// TwinCAT 3 PLC project plc_polycap_01
// ProgramVersion: 3.1.4023.0
// libraries:
//   LCLS General, * (SLAC)
//   lcls-twincat-motion, * (SLAC)
//   Tc2_Standard, * (Beckhoff Automation GmbH)
//   Tc2_System, * (Beckhoff Automation GmbH)
//   Tc3_Module, * (Beckhoff Automation GmbH)
// project tree:
//   GVLs/ Main.TcGVL
//   / PlcTask.TcTTO (not stored)
//   POUs/ PRG_SPEC.TcPOU
// real-time tasks:
//   TASK PlcTask: cycle T#10ms, priority 20, ADS port 350
// motion (NC):
//   TASK NC-Task 1 SAF: cycle T#2ms, priority 4, ADS port 501
//   TASK NC-Task 1 SVB: cycle T#10ms, priority 8, ADS port 511
//   AXIS Axis 1 POLYCAP-DET-Z (id 1)
//     Velo: Maximum=5
//     OtherSettings: AllowMotionCmdToSlave=true
//     encoder EncType=4
//       EncPara: ScaleFactorNumerator=7.8125e-05, MaxCount=#x0000ffff
//         Inc: RefSoftSyncMask=#x0000ffff
//     drive DrvType=24
//       Analog: VeloReferenz=10, TorqueSetpointScale=10, ScaleFactorActTorque=0.1
//       TimeComp: TaskDelayCycles=1
//     controller CtrType=1
//       CtrPara: PriorControlFactor=1
//         Observer: BandWidth=20
//   AXIS Axis 2 POLYCAP-CRY-N-SWI (id 2)
//     Velo: Maximum=5
//     OtherSettings: AllowMotionCmdToSlave=true
//     encoder EncType=4
//       EncPara: ScaleFactorNumerator=5.234375e-05, MaxCount=#x0000ffff
//         Inc: RefSoftSyncMask=#x0000ffff
//     drive DrvType=24
//       Analog: VeloReferenz=6.7, TorqueSetpointScale=10, ScaleFactorActTorque=0.1
//       TimeComp: TaskDelayCycles=1
//     controller CtrType=1
//       CtrPara: PriorControlFactor=1
//         Observer: BandWidth=20
//   AXIS Axis 3 POLYCAP-CRY-N-X (id 3)
//     Velo: Maximum=5
//     OtherSettings: AllowMotionCmdToSlave=true
//     encoder EncType=4
//       EncPara: ScaleFactorNumerator=7.8125e-05, MaxCount=#x0000ffff
//         Inc: RefSoftSyncMask=#x0000ffff
//     drive DrvType=24
//       Analog: VeloReferenz=10, TorqueSetpointScale=10, ScaleFactorActTorque=0.1
//       TimeComp: TaskDelayCycles=1
//     controller CtrType=1
//       CtrPara: PriorControlFactor=1
//         Observer: BandWidth=20
//   AXIS Axis 4 POLYCAP-CRY-N-ROT (id 4)
//     Velo: Maximum=5
//     OtherSettings: AllowMotionCmdToSlave=true
//     encoder EncType=4
//       EncPara: ScaleFactorNumerator=0.00015625, MaxCount=#x0000ffff
//         Inc: RefSoftSyncMask=#x0000ffff
//     drive DrvType=24
//       Analog: VeloReferenz=20, TorqueSetpointScale=10, ScaleFactorActTorque=0.1
//       TimeComp: TaskDelayCycles=1
//     controller CtrType=1
//       CtrPara: PriorControlFactor=1
//         Observer: BandWidth=20
//   AXIS Axis 5 POLYCAP-CRY-N-Y (id 5)
//     Velo: Maximum=5
//     OtherSettings: AllowMotionCmdToSlave=true
//     encoder EncType=4
//       EncPara: ScaleFactorNumerator=7.8125e-05, MaxCount=#x0000ffff
//         Inc: RefSoftSyncMask=#x0000ffff
//     drive DrvType=24
//       Analog: VeloReferenz=10, TorqueSetpointScale=10, ScaleFactorActTorque=0.1
//       TimeComp: TaskDelayCycles=1
//     controller CtrType=1
//       CtrPara: PriorControlFactor=1
//         Observer: BandWidth=20
//   AXIS Axis 6 POLYCAP-PC-N-X (id 6)
//     Velo: Maximum=5
//     OtherSettings: AllowMotionCmdToSlave=true
//     encoder EncType=4
//       EncPara: ScaleFactorNumerator=3.90625e-05, MaxCount=#x0000ffff
//         Inc: RefSoftSyncMask=#x0000ffff
//     drive DrvType=24
//       Analog: VeloReferenz=5, TorqueSetpointScale=10, ScaleFactorActTorque=0.1
//       TimeComp: TaskDelayCycles=1
//     controller CtrType=1
//       CtrPara: PriorControlFactor=1
//         Observer: BandWidth=20
//   AXIS Axis 7 POLYCAP-PC-N-Z (id 7)
//     Velo: Maximum=5
//     OtherSettings: AllowMotionCmdToSlave=true
//     encoder EncType=4
//       EncPara: ScaleFactorNumerator=1.953125e-05, MaxCount=#x0000ffff
//         Inc: RefSoftSyncMask=#x0000ffff
//     drive DrvType=24
//       Analog: VeloReferenz=2.5, TorqueSetpointScale=10, ScaleFactorActTorque=0.1
//       TimeComp: TaskDelayCycles=1
//     controller CtrType=1
//       CtrPara: PriorControlFactor=1
//         Observer: BandWidth=20
//   AXIS Axis 8 POLYCAP-PC-N-Y (id 8)
//     Velo: Maximum=5
//     OtherSettings: AllowMotionCmdToSlave=true
//     encoder EncType=4
//       EncPara: ScaleFactorNumerator=3.90625e-05, MaxCount=#x0000ffff
//         Inc: RefSoftSyncMask=#x0000ffff
//     drive DrvType=24
//       Analog: VeloReferenz=5, TorqueSetpointScale=10, ScaleFactorActTorque=0.1
//       TimeComp: TaskDelayCycles=1
//     controller CtrType=1
//       CtrPara: PriorControlFactor=1
//         Observer: BandWidth=20
//   AXIS Axis 9 POLYCAP-CRY-S-SWI (id 9)
//     Velo: Maximum=5
//     OtherSettings: AllowMotionCmdToSlave=true
//     encoder EncType=4
//       EncPara: ScaleFactorNumerator=5.234375e-05, MaxCount=#x0000ffff
//         Inc: RefSoftSyncMask=#x0000ffff
//     drive DrvType=24
//       Analog: VeloReferenz=6.7, TorqueSetpointScale=10, ScaleFactorActTorque=0.1
//       TimeComp: TaskDelayCycles=1
//     controller CtrType=1
//       CtrPara: PriorControlFactor=1
//         Observer: BandWidth=20
//   AXIS Axis 10 POLYCAP-CRY-S-X (id 10)
//     Velo: Maximum=5
//     OtherSettings: AllowMotionCmdToSlave=true
//     encoder EncType=4
//       EncPara: ScaleFactorNumerator=7.8125e-05, MaxCount=#x0000ffff
//         Inc: RefSoftSyncMask=#x0000ffff
//     drive DrvType=24
//       Analog: VeloReferenz=10, TorqueSetpointScale=10, ScaleFactorActTorque=0.1
//       TimeComp: TaskDelayCycles=1
//     controller CtrType=1
//       CtrPara: PriorControlFactor=1
//         Observer: BandWidth=20
//   AXIS Axis 11 POLYCAP-CRY-M-SWI (id 11)
//     Velo: Maximum=5
//     OtherSettings: AllowMotionCmdToSlave=true
//     encoder EncType=4
//       EncPara: ScaleFactorNumerator=5.234375e-05, MaxCount=#x0000ffff
//         Inc: RefSoftSyncMask=#x0000ffff
//     drive DrvType=24
//       Analog: VeloReferenz=6.7, TorqueSetpointScale=10, ScaleFactorActTorque=0.1
//       TimeComp: TaskDelayCycles=1
//     controller CtrType=1
//       CtrPara: PriorControlFactor=1
//         Observer: BandWidth=20
//   AXIS Axis 12 POLYCAP-CRY-M-X (id 12)
//     Velo: Maximum=5
//     OtherSettings: AllowMotionCmdToSlave=true
//     encoder EncType=4
//       EncPara: ScaleFactorNumerator=7.8125e-05, MaxCount=#x0000ffff
//         Inc: RefSoftSyncMask=#x0000ffff
//     drive DrvType=24
//       Analog: VeloReferenz=10, TorqueSetpointScale=10, ScaleFactorActTorque=0.1
//       TimeComp: TaskDelayCycles=1
//     controller CtrType=1
//       CtrPara: PriorControlFactor=1
//         Observer: BandWidth=20
//   AXIS Axis 13 POLYCAP-CRY-S-ROT (id 13)
//     Velo: Maximum=5
//     OtherSettings: AllowMotionCmdToSlave=true
//     encoder EncType=4
//       EncPara: ScaleFactorNumerator=0.00015625, MaxCount=#x0000ffff
//         Inc: RefSoftSyncMask=#x0000ffff
//     drive DrvType=24
//       Analog: VeloReferenz=20, TorqueSetpointScale=10, ScaleFactorActTorque=0.1
//       TimeComp: TaskDelayCycles=1
//     controller CtrType=1
//       CtrPara: PriorControlFactor=1
//         Observer: BandWidth=20
//   AXIS Axis 14 POLYCAP-CRY-S-Y (id 14)
//     Velo: Maximum=5
//     OtherSettings: AllowMotionCmdToSlave=true
//     encoder EncType=4
//       EncPara: ScaleFactorNumerator=7.8125e-05, MaxCount=#x0000ffff
//         Inc: RefSoftSyncMask=#x0000ffff
//     drive DrvType=24
//       Analog: VeloReferenz=10, TorqueSetpointScale=10, ScaleFactorActTorque=0.1
//       TimeComp: TaskDelayCycles=1
//     controller CtrType=1
//       CtrPara: PriorControlFactor=1
//         Observer: BandWidth=20
//   AXIS Axis 15 POLYCAP-CRY-M-ROT (id 15)
//     Velo: Maximum=5
//     OtherSettings: AllowMotionCmdToSlave=true
//     encoder EncType=4
//       EncPara: ScaleFactorNumerator=0.00015625, MaxCount=#x0000ffff
//         Inc: RefSoftSyncMask=#x0000ffff
//     drive DrvType=24
//       Analog: VeloReferenz=20, TorqueSetpointScale=10, ScaleFactorActTorque=0.1
//       TimeComp: TaskDelayCycles=1
//     controller CtrType=1
//       CtrPara: PriorControlFactor=1
//         Observer: BandWidth=20
//   AXIS Axis 16 POLYCAP-CRY-M-Y (id 16)
//     Velo: Maximum=5
//     OtherSettings: AllowMotionCmdToSlave=true
//     encoder EncType=4
//       EncPara: ScaleFactorNumerator=7.8125e-05, MaxCount=#x0000ffff
//         Inc: RefSoftSyncMask=#x0000ffff
//     drive DrvType=24
//       Analog: VeloReferenz=10, TorqueSetpointScale=10, ScaleFactorActTorque=0.1
//       TimeComp: TaskDelayCycles=1
//     controller CtrType=1
//       CtrPara: PriorControlFactor=1
//         Observer: BandWidth=20
//   AXIS Axis 17 POLYCAP-PC-S-X (id 17)
//     Velo: Maximum=5
//     OtherSettings: AllowMotionCmdToSlave=true
//     encoder EncType=4
//       EncPara: ScaleFactorNumerator=3.90625e-05, MaxCount=#x0000ffff
//         Inc: RefSoftSyncMask=#x0000ffff
//     drive DrvType=24
//       Analog: VeloReferenz=5, TorqueSetpointScale=10, ScaleFactorActTorque=0.1
//       TimeComp: TaskDelayCycles=1
//     controller CtrType=1
//       CtrPara: PriorControlFactor=1
//         Observer: BandWidth=20
//   AXIS Axis 18 POLYCAP-PC-S-Z (id 18)
//     Velo: Maximum=5
//     OtherSettings: AllowMotionCmdToSlave=true
//     encoder EncType=4
//       EncPara: ScaleFactorNumerator=1.953125e-05, MaxCount=#x0000ffff
//         Inc: RefSoftSyncMask=#x0000ffff
//     drive DrvType=24
//       Analog: VeloReferenz=2.5, TorqueSetpointScale=10, ScaleFactorActTorque=0.1
//       TimeComp: TaskDelayCycles=1
//     controller CtrType=1
//       CtrPara: PriorControlFactor=1
//         Observer: BandWidth=20
//   AXIS Axis 19 POLYCAP-PC-M-X (id 19)
//     Velo: Maximum=5
//     OtherSettings: AllowMotionCmdToSlave=true
//     encoder EncType=4
//       EncPara: ScaleFactorNumerator=3.90625e-05, MaxCount=#x0000ffff
//         Inc: RefSoftSyncMask=#x0000ffff
//     drive DrvType=24
//       Analog: VeloReferenz=5, TorqueSetpointScale=10, ScaleFactorActTorque=0.1
//       TimeComp: TaskDelayCycles=1
//     controller CtrType=1
//       CtrPara: PriorControlFactor=1
//         Observer: BandWidth=20
//   AXIS Axis 20 POLYCAP-PC-M-Z (id 20)
//     Velo: Maximum=5
//     OtherSettings: AllowMotionCmdToSlave=true
//     encoder EncType=4
//       EncPara: ScaleFactorNumerator=1.953125e-05, MaxCount=#x0000ffff
//         Inc: RefSoftSyncMask=#x0000ffff
//     drive DrvType=24
//       Analog: VeloReferenz=2.5, TorqueSetpointScale=10, ScaleFactorActTorque=0.1
//       TimeComp: TaskDelayCycles=1
//     controller CtrType=1
//       CtrPara: PriorControlFactor=1
//         Observer: BandWidth=20
//   AXIS Axis 21 POLYCAP-PC-S-Y (id 21)
//     Velo: Maximum=5
//     OtherSettings: AllowMotionCmdToSlave=true
//     encoder EncType=4
//       EncPara: ScaleFactorNumerator=3.90625e-05, MaxCount=#x0000ffff
//         Inc: RefSoftSyncMask=#x0000ffff
//     drive DrvType=24
//       Analog: VeloReferenz=5, TorqueSetpointScale=10, ScaleFactorActTorque=0.1
//       TimeComp: TaskDelayCycles=1
//     controller CtrType=1
//       CtrPara: PriorControlFactor=1
//         Observer: BandWidth=20
//   AXIS Axis 22 POLYCAP-PC-M-Y (id 22)
//     Velo: Maximum=5
//     OtherSettings: AllowMotionCmdToSlave=true
//     encoder EncType=4
//       EncPara: ScaleFactorNumerator=3.90625e-05, MaxCount=#x0000ffff
//         Inc: RefSoftSyncMask=#x0000ffff
//     drive DrvType=24
//       Analog: VeloReferenz=5, TorqueSetpointScale=10, ScaleFactorActTorque=0.1
//       TimeComp: TaskDelayCycles=1
//     controller CtrType=1
//       CtrPara: PriorControlFactor=1
//         Observer: BandWidth=20
// I/O:
//   DEVICE Device 1 (EtherCAT), AmsNetId 172.21.148.88.2.1
//     Term 1 (EK1200) [EK1200-5000 EtherCAT Power supply (2A E-Bus)]
//       POLYCAP1-EL7031-E1 [EL7031 1Ch. Stepper motor output stage (24V, 1.5A)]
//       Term 3 (EL6070) [EL6070 1Ch. Licensing-Terminal]
//       Term 4 (EL7031) [EL7031 1Ch. Stepper motor output stage (24V, 1.5A)]
//       POLYCAP1-EL1088-E4 [EL1088 8Ch. Dig. Input 24V, 3ms, negative]
//       Term 6 (EL7031) [EL7031 1Ch. Stepper motor output stage (24V, 1.5A)]
//       Term 7 (EL7031) [EL7031 1Ch. Stepper motor output stage (24V, 1.5A)]
//       Term 8 (EL7031) [EL7031 1Ch. Stepper motor output stage (24V, 1.5A)]
//       Term 9 (EL7031) [EL7031 1Ch. Stepper motor output stage (24V, 1.5A)]
//       POLYCAP1-EL1088-E9 [EL1088 8Ch. Dig. Input 24V, 3ms, negative]
//       Term 11 (EK1122) [EK1122 2 port EtherCAT junction]
//         Term 12 (EK1100) [EK1100 EtherCAT Coupler (2A E-Bus)]
//           Term 13 (EL7031) [EL7031 1Ch. Stepper motor output stage (24V, 1.5A)]
//           Term 14 (EL7031) [EL7031 1Ch. Stepper motor output stage (24V, 1.5A)]
//           POLYCAP2-EL1088-E3 [EL1088 8Ch. Dig. Input 24V, 3ms, negative]
//           Term 16 (EL7031) [EL7031 1Ch. Stepper motor output stage (24V, 1.5A)]
//           Term 17 (EL7031) [EL7031 1Ch. Stepper motor output stage (24V, 1.5A)]
//           Term 18 (EL7031) [EL7031 1Ch. Stepper motor output stage (24V, 1.5A)]
//           Term 19 (EL7031) [EL7031 1Ch. Stepper motor output stage (24V, 1.5A)]
//           POLYCAP2-EL1088-E8 [EL1088 8Ch. Dig. Input 24V, 3ms, negative]
//           Term 21 (EL7031) [EL7031 1Ch. Stepper motor output stage (24V, 1.5A)]
//           Term 22 (EL7031) [EL7031 1Ch. Stepper motor output stage (24V, 1.5A)]
//           Term 23 (EL9410) [EL9410 E-Bus Power Supplier  (Diagnostics)]
//           Term 24 (EL7031) [EL7031 1Ch. Stepper motor output stage (24V, 1.5A)]
//           Term 25 (EL7031) [EL7031 1Ch. Stepper motor output stage (24V, 1.5A)]
//           POLYCAP2-EL1088-E14 [EL1088 8Ch. Dig. Input 24V, 3ms, negative]
//           Term 27 (EL7031) [EL7031 1Ch. Stepper motor output stage (24V, 1.5A)]
//           Term 28 (EL7031) [EL7031 1Ch. Stepper motor output stage (24V, 1.5A)]
//           Term 29 (EL7031) [EL7031 1Ch. Stepper motor output stage (24V, 1.5A)]
//           Term 30 (EL7031) [EL7031 1Ch. Stepper motor output stage (24V, 1.5A)]
//           POLYCAP2-EL1088-E19 [EL1088 8Ch. Dig. Input 24V, 3ms, negative]
//           Term 32 (EL7031) [EL7031 1Ch. Stepper motor output stage (24V, 1.5A)]
//           Term 33 (EL7031) [EL7031 1Ch. Stepper motor output stage (24V, 1.5A)]
//           Term 34 (EL9011)
// variable links:
//   (this object) <-> Device 1 (EtherCAT)/Term 1 (EK1200)/POLYCAP1-EL7031-E1
//     Drive/Inputs/In/nState1 @bit 3 <-> STM Status/Status/Error
//     Drive/Inputs/In/nState1 @bit 5 <-> STM Status/Status/Moving negative
//     Drive/Inputs/In/nState1 @bit 4 <-> STM Status/Status/Moving positive
//     Drive/Inputs/In/nState1 @bit 1 <-> STM Status/Status/Ready
//     Drive/Inputs/In/nState1 <-> STM Status/Status/Ready to enable
//     Drive/Inputs/In/nState1 @bit 6 <-> STM Status/Status/Torque reduced
//     Drive/Inputs/In/nState1 @bit 2 <-> STM Status/Status/Warning
//     Drive/Inputs/In/nState2 @bit 3 <-> STM Status/Status/Digital input 1
//     Drive/Inputs/In/nState2 @bit 4 <-> STM Status/Status/Digital input 2
//     Drive/Inputs/In/nState2 @bit 5 <-> STM Status/Status/Sync error
//     Drive/Inputs/In/nState2 @bit 7 <-> STM Status/Status/TxPDO Toggle
//     Drive/Inputs/In/nState4 @bit 1 <-> WcState/InputToggle
//     Drive/Inputs/In/nState4 <-> WcState/WcState
//     Drive/Outputs/Out/nCtrl1 <-> STM Control/Control/Enable
//     Drive/Outputs/Out/nCtrl1 @bit 2 <-> STM Control/Control/Reduce torque
//     Drive/Outputs/Out/nCtrl1 @bit 1 <-> STM Control/Control/Reset
//     Drive/Outputs/Out/nDataOut2[0] <-> STM Velocity/Velocity
//     Enc/Inputs/In/nDataIn1[0] <-> ENC Status compact/Counter value
//     Enc/Inputs/In/nDataIn2[0] <-> ENC Status compact/Latch value
//     Enc/Inputs/In/nState1 @bit 4 <-> ENC Status compact/Status/Counter overflow
//     Enc/Inputs/In/nState1 @bit 3 <-> ENC Status compact/Status/Counter underflow
//     Enc/Inputs/In/nState1 @bit 1 <-> ENC Status compact/Status/Latch extern valid
//     Enc/Inputs/In/nState1 @bit 2 <-> ENC Status compact/Status/Set counter done
//     Enc/Inputs/In/nState2 @bit 4 <-> ENC Status compact/Status/Status of extern latch
//     Enc/Inputs/In/nState2 @bit 5 <-> ENC Status compact/Status/Sync error
//     Enc/Inputs/In/nState2 @bit 7 <-> ENC Status compact/Status/TxPDO Toggle
//     Enc/Inputs/In/nState4 @bit 1 <-> WcState/InputToggle
//     Enc/Inputs/In/nState4 <-> WcState/WcState
//     Enc/Outputs/Out/nCtrl1 @bit 3 <-> ENC Control compact/Control/Enable latch extern on negative edge
//     Enc/Outputs/Out/nCtrl1 @bit 1 <-> ENC Control compact/Control/Enable latch extern on positive edge
//     Enc/Outputs/Out/nCtrl1 @bit 2 <-> ENC Control compact/Control/Set counter
//     Enc/Outputs/Out/nDataOut1[0] <-> ENC Control compact/Set counter value
//   (this object) <-> Device 1 (EtherCAT)/Term 1 (EK1200)/Term 4 (EL7031)
//     Drive/Inputs/In/nState1 @bit 3 <-> STM Status/Status/Error
//     Drive/Inputs/In/nState1 @bit 5 <-> STM Status/Status/Moving negative
//     Drive/Inputs/In/nState1 @bit 4 <-> STM Status/Status/Moving positive
//     Drive/Inputs/In/nState1 @bit 1 <-> STM Status/Status/Ready
//     Drive/Inputs/In/nState1 <-> STM Status/Status/Ready to enable
//     Drive/Inputs/In/nState1 @bit 6 <-> STM Status/Status/Torque reduced
//     Drive/Inputs/In/nState1 @bit 2 <-> STM Status/Status/Warning
//     Drive/Inputs/In/nState2 @bit 3 <-> STM Status/Status/Digital input 1
//     Drive/Inputs/In/nState2 @bit 4 <-> STM Status/Status/Digital input 2
//     Drive/Inputs/In/nState2 @bit 5 <-> STM Status/Status/Sync error
//     Drive/Inputs/In/nState2 @bit 7 <-> STM Status/Status/TxPDO Toggle
//     Drive/Inputs/In/nState4 @bit 1 <-> WcState/InputToggle
//     Drive/Inputs/In/nState4 <-> WcState/WcState
//     Drive/Outputs/Out/nCtrl1 <-> STM Control/Control/Enable
//     Drive/Outputs/Out/nCtrl1 @bit 2 <-> STM Control/Control/Reduce torque
//     Drive/Outputs/Out/nCtrl1 @bit 1 <-> STM Control/Control/Reset
//     Drive/Outputs/Out/nDataOut2[0] <-> STM Velocity/Velocity
//     Enc/Inputs/In/nDataIn1[0] <-> ENC Status compact/Counter value
//     Enc/Inputs/In/nDataIn2[0] <-> ENC Status compact/Latch value
//     Enc/Inputs/In/nState1 @bit 4 <-> ENC Status compact/Status/Counter overflow
//     Enc/Inputs/In/nState1 @bit 3 <-> ENC Status compact/Status/Counter underflow
//     Enc/Inputs/In/nState1 @bit 1 <-> ENC Status compact/Status/Latch extern valid
//     Enc/Inputs/In/nState1 @bit 2 <-> ENC Status compact/Status/Set counter done
//     Enc/Inputs/In/nState2 @bit 4 <-> ENC Status compact/Status/Status of extern latch
//     Enc/Inputs/In/nState2 @bit 5 <-> ENC Status compact/Status/Sync error
//     Enc/Inputs/In/nState2 @bit 7 <-> ENC Status compact/Status/TxPDO Toggle
//     Enc/Inputs/In/nState4 @bit 1 <-> WcState/InputToggle
//     Enc/Inputs/In/nState4 <-> WcState/WcState
//     Enc/Outputs/Out/nCtrl1 @bit 3 <-> ENC Control compact/Control/Enable latch extern on negative edge
//     Enc/Outputs/Out/nCtrl1 @bit 1 <-> ENC Control compact/Control/Enable latch extern on positive edge
//     Enc/Outputs/Out/nCtrl1 @bit 2 <-> ENC Control compact/Control/Set counter
//     Enc/Outputs/Out/nDataOut1[0] <-> ENC Control compact/Set counter value
//   (this object) <-> Device 1 (EtherCAT)/Term 1 (EK1200)/Term 6 (EL7031)
//     Drive/Inputs/In/nState1 @bit 3 <-> STM Status/Status/Error
//     Drive/Inputs/In/nState1 @bit 5 <-> STM Status/Status/Moving negative
//     Drive/Inputs/In/nState1 @bit 4 <-> STM Status/Status/Moving positive
//     Drive/Inputs/In/nState1 @bit 1 <-> STM Status/Status/Ready
//     Drive/Inputs/In/nState1 <-> STM Status/Status/Ready to enable
//     Drive/Inputs/In/nState1 @bit 6 <-> STM Status/Status/Torque reduced
//     Drive/Inputs/In/nState1 @bit 2 <-> STM Status/Status/Warning
//     Drive/Inputs/In/nState2 @bit 3 <-> STM Status/Status/Digital input 1
//     Drive/Inputs/In/nState2 @bit 4 <-> STM Status/Status/Digital input 2
//     Drive/Inputs/In/nState2 @bit 5 <-> STM Status/Status/Sync error
//     Drive/Inputs/In/nState2 @bit 7 <-> STM Status/Status/TxPDO Toggle
//     Drive/Inputs/In/nState4 @bit 1 <-> WcState/InputToggle
//     Drive/Inputs/In/nState4 <-> WcState/WcState
//     Drive/Outputs/Out/nCtrl1 <-> STM Control/Control/Enable
//     Drive/Outputs/Out/nCtrl1 @bit 2 <-> STM Control/Control/Reduce torque
//     Drive/Outputs/Out/nCtrl1 @bit 1 <-> STM Control/Control/Reset
//     Drive/Outputs/Out/nDataOut2[0] <-> STM Velocity/Velocity
//     Enc/Inputs/In/nDataIn1[0] <-> ENC Status compact/Counter value
//     Enc/Inputs/In/nDataIn2[0] <-> ENC Status compact/Latch value
//     Enc/Inputs/In/nState1 @bit 4 <-> ENC Status compact/Status/Counter overflow
//     Enc/Inputs/In/nState1 @bit 3 <-> ENC Status compact/Status/Counter underflow
//     Enc/Inputs/In/nState1 @bit 1 <-> ENC Status compact/Status/Latch extern valid
//     Enc/Inputs/In/nState1 @bit 2 <-> ENC Status compact/Status/Set counter done
//     Enc/Inputs/In/nState2 @bit 4 <-> ENC Status compact/Status/Status of extern latch
//     Enc/Inputs/In/nState2 @bit 5 <-> ENC Status compact/Status/Sync error
//     Enc/Inputs/In/nState2 @bit 7 <-> ENC Status compact/Status/TxPDO Toggle
//     Enc/Inputs/In/nState4 @bit 1 <-> WcState/InputToggle
//     Enc/Inputs/In/nState4 <-> WcState/WcState
//     Enc/Outputs/Out/nCtrl1 @bit 3 <-> ENC Control compact/Control/Enable latch extern on negative edge
//     Enc/Outputs/Out/nCtrl1 @bit 1 <-> ENC Control compact/Control/Enable latch extern on positive edge
//     Enc/Outputs/Out/nCtrl1 @bit 2 <-> ENC Control compact/Control/Set counter
//     Enc/Outputs/Out/nDataOut1[0] <-> ENC Control compact/Set counter value
//   (this object) <-> Device 1 (EtherCAT)/Term 1 (EK1200)/Term 7 (EL7031)
//     Drive/Inputs/In/nState1 @bit 3 <-> STM Status/Status/Error
//     Drive/Inputs/In/nState1 @bit 5 <-> STM Status/Status/Moving negative
//     Drive/Inputs/In/nState1 @bit 4 <-> STM Status/Status/Moving positive
//     Drive/Inputs/In/nState1 @bit 1 <-> STM Status/Status/Ready
//     Drive/Inputs/In/nState1 <-> STM Status/Status/Ready to enable
//     Drive/Inputs/In/nState1 @bit 6 <-> STM Status/Status/Torque reduced
//     Drive/Inputs/In/nState1 @bit 2 <-> STM Status/Status/Warning
//     Drive/Inputs/In/nState2 @bit 3 <-> STM Status/Status/Digital input 1
//     Drive/Inputs/In/nState2 @bit 4 <-> STM Status/Status/Digital input 2
//     Drive/Inputs/In/nState2 @bit 5 <-> STM Status/Status/Sync error
//     Drive/Inputs/In/nState2 @bit 7 <-> STM Status/Status/TxPDO Toggle
//     Drive/Inputs/In/nState4 @bit 1 <-> WcState/InputToggle
//     Drive/Inputs/In/nState4 <-> WcState/WcState
//     Drive/Outputs/Out/nCtrl1 <-> STM Control/Control/Enable
//     Drive/Outputs/Out/nCtrl1 @bit 2 <-> STM Control/Control/Reduce torque
//     Drive/Outputs/Out/nCtrl1 @bit 1 <-> STM Control/Control/Reset
//     Drive/Outputs/Out/nDataOut2[0] <-> STM Velocity/Velocity
//     Enc/Inputs/In/nDataIn1[0] <-> ENC Status compact/Counter value
//     Enc/Inputs/In/nDataIn2[0] <-> ENC Status compact/Latch value
//     Enc/Inputs/In/nState1 @bit 4 <-> ENC Status compact/Status/Counter overflow
//     Enc/Inputs/In/nState1 @bit 3 <-> ENC Status compact/Status/Counter underflow
//     Enc/Inputs/In/nState1 @bit 1 <-> ENC Status compact/Status/Latch extern valid
//     Enc/Inputs/In/nState1 @bit 2 <-> ENC Status compact/Status/Set counter done
//     Enc/Inputs/In/nState2 @bit 4 <-> ENC Status compact/Status/Status of extern latch
//     Enc/Inputs/In/nState2 @bit 5 <-> ENC Status compact/Status/Sync error
//     Enc/Inputs/In/nState2 @bit 7 <-> ENC Status compact/Status/TxPDO Toggle
//     Enc/Inputs/In/nState4 @bit 1 <-> WcState/InputToggle
//     Enc/Inputs/In/nState4 <-> WcState/WcState
//     Enc/Outputs/Out/nCtrl1 @bit 3 <-> ENC Control compact/Control/Enable latch extern on negative edge
//     Enc/Outputs/Out/nCtrl1 @bit 1 <-> ENC Control compact/Control/Enable latch extern on positive edge
//     Enc/Outputs/Out/nCtrl1 @bit 2 <-> ENC Control compact/Control/Set counter
//     Enc/Outputs/Out/nDataOut1[0] <-> ENC Control compact/Set counter value
//   (this object) <-> Device 1 (EtherCAT)/Term 1 (EK1200)/Term 8 (EL7031)
//     Drive/Inputs/In/nState1 @bit 3 <-> STM Status/Status/Error
//     Drive/Inputs/In/nState1 @bit 5 <-> STM Status/Status/Moving negative
//     Drive/Inputs/In/nState1 @bit 4 <-> STM Status/Status/Moving positive
//     Drive/Inputs/In/nState1 @bit 1 <-> STM Status/Status/Ready
//     Drive/Inputs/In/nState1 <-> STM Status/Status/Ready to enable
//     Drive/Inputs/In/nState1 @bit 6 <-> STM Status/Status/Torque reduced
//     Drive/Inputs/In/nState1 @bit 2 <-> STM Status/Status/Warning
//     Drive/Inputs/In/nState2 @bit 3 <-> STM Status/Status/Digital input 1
//     Drive/Inputs/In/nState2 @bit 4 <-> STM Status/Status/Digital input 2
//     Drive/Inputs/In/nState2 @bit 5 <-> STM Status/Status/Sync error
//     Drive/Inputs/In/nState2 @bit 7 <-> STM Status/Status/TxPDO Toggle
//     Drive/Inputs/In/nState4 @bit 1 <-> WcState/InputToggle
//     Drive/Inputs/In/nState4 <-> WcState/WcState
//     Drive/Outputs/Out/nCtrl1 <-> STM Control/Control/Enable
//     Drive/Outputs/Out/nCtrl1 @bit 2 <-> STM Control/Control/Reduce torque
//     Drive/Outputs/Out/nCtrl1 @bit 1 <-> STM Control/Control/Reset
//     Drive/Outputs/Out/nDataOut2[0] <-> STM Velocity/Velocity
//     Enc/Inputs/In/nDataIn1[0] <-> ENC Status compact/Counter value
//     Enc/Inputs/In/nDataIn2[0] <-> ENC Status compact/Latch value
//     Enc/Inputs/In/nState1 @bit 4 <-> ENC Status compact/Status/Counter overflow
//     Enc/Inputs/In/nState1 @bit 3 <-> ENC Status compact/Status/Counter underflow
//     Enc/Inputs/In/nState1 @bit 1 <-> ENC Status compact/Status/Latch extern valid
//     Enc/Inputs/In/nState1 @bit 2 <-> ENC Status compact/Status/Set counter done
//     Enc/Inputs/In/nState2 @bit 4 <-> ENC Status compact/Status/Status of extern latch
//     Enc/Inputs/In/nState2 @bit 5 <-> ENC Status compact/Status/Sync error
//     Enc/Inputs/In/nState2 @bit 7 <-> ENC Status compact/Status/TxPDO Toggle
//     Enc/Inputs/In/nState4 @bit 1 <-> WcState/InputToggle
//     Enc/Inputs/In/nState4 <-> WcState/WcState
//     Enc/Outputs/Out/nCtrl1 @bit 3 <-> ENC Control compact/Control/Enable latch extern on negative edge
//     Enc/Outputs/Out/nCtrl1 @bit 1 <-> ENC Control compact/Control/Enable latch extern on positive edge
//     Enc/Outputs/Out/nCtrl1 @bit 2 <-> ENC Control compact/Control/Set counter
//     Enc/Outputs/Out/nDataOut1[0] <-> ENC Control compact/Set counter value
//   (this object) <-> Device 1 (EtherCAT)/Term 1 (EK1200)/Term 9 (EL7031)
//     Drive/Inputs/In/nState1 @bit 3 <-> STM Status/Status/Error
//     Drive/Inputs/In/nState1 @bit 5 <-> STM Status/Status/Moving negative
//     Drive/Inputs/In/nState1 @bit 4 <-> STM Status/Status/Moving positive
//     Drive/Inputs/In/nState1 @bit 1 <-> STM Status/Status/Ready
//     Drive/Inputs/In/nState1 <-> STM Status/Status/Ready to enable
//     Drive/Inputs/In/nState1 @bit 6 <-> STM Status/Status/Torque reduced
//     Drive/Inputs/In/nState1 @bit 2 <-> STM Status/Status/Warning
//     Drive/Inputs/In/nState2 @bit 3 <-> STM Status/Status/Digital input 1
//     Drive/Inputs/In/nState2 @bit 4 <-> STM Status/Status/Digital input 2
//     Drive/Inputs/In/nState2 @bit 5 <-> STM Status/Status/Sync error
//     Drive/Inputs/In/nState2 @bit 7 <-> STM Status/Status/TxPDO Toggle
//     Drive/Inputs/In/nState4 @bit 1 <-> WcState/InputToggle
//     Drive/Inputs/In/nState4 <-> WcState/WcState
//     Drive/Outputs/Out/nCtrl1 <-> STM Control/Control/Enable
//     Drive/Outputs/Out/nCtrl1 @bit 2 <-> STM Control/Control/Reduce torque
//     Drive/Outputs/Out/nCtrl1 @bit 1 <-> STM Control/Control/Reset
//     Drive/Outputs/Out/nDataOut2[0] <-> STM Velocity/Velocity
//     Enc/Inputs/In/nDataIn1[0] <-> ENC Status compact/Counter value
//     Enc/Inputs/In/nDataIn2[0] <-> ENC Status compact/Latch value
//     Enc/Inputs/In/nState1 @bit 4 <-> ENC Status compact/Status/Counter overflow
//     Enc/Inputs/In/nState1 @bit 3 <-> ENC Status compact/Status/Counter underflow
//     Enc/Inputs/In/nState1 @bit 1 <-> ENC Status compact/Status/Latch extern valid
//     Enc/Inputs/In/nState1 @bit 2 <-> ENC Status compact/Status/Set counter done
//     Enc/Inputs/In/nState2 @bit 4 <-> ENC Status compact/Status/Status of extern latch
//     Enc/Inputs/In/nState2 @bit 5 <-> ENC Status compact/Status/Sync error
//     Enc/Inputs/In/nState2 @bit 7 <-> ENC Status compact/Status/TxPDO Toggle
//     Enc/Inputs/In/nState4 @bit 1 <-> WcState/InputToggle
//     Enc/Inputs/In/nState4 <-> WcState/WcState
//     Enc/Outputs/Out/nCtrl1 @bit 3 <-> ENC Control compact/Control/Enable latch extern on negative edge
//     Enc/Outputs/Out/nCtrl1 @bit 1 <-> ENC Control compact/Control/Enable latch extern on positive edge
//     Enc/Outputs/Out/nCtrl1 @bit 2 <-> ENC Control compact/Control/Set counter
//     Enc/Outputs/Out/nDataOut1[0] <-> ENC Control compact/Set counter value
//   (this object) <-> Device 1 (EtherCAT)/Term 1 (EK1200)/Term 11 (EK1122)/Term 12 (EK1100)/Term 13 (EL7031)
//     Drive/Inputs/In/nState1 @bit 3 <-> STM Status/Status/Error
//     Drive/Inputs/In/nState1 @bit 5 <-> STM Status/Status/Moving negative
//     Drive/Inputs/In/nState1 @bit 4 <-> STM Status/Status/Moving positive
//     Drive/Inputs/In/nState1 @bit 1 <-> STM Status/Status/Ready
//     Drive/Inputs/In/nState1 <-> STM Status/Status/Ready to enable
//     Drive/Inputs/In/nState1 @bit 6 <-> STM Status/Status/Torque reduced
//     Drive/Inputs/In/nState1 @bit 2 <-> STM Status/Status/Warning
//     Drive/Inputs/In/nState2 @bit 3 <-> STM Status/Status/Digital input 1
//     Drive/Inputs/In/nState2 @bit 4 <-> STM Status/Status/Digital input 2
//     Drive/Inputs/In/nState2 @bit 5 <-> STM Status/Status/Sync error
//     Drive/Inputs/In/nState2 @bit 7 <-> STM Status/Status/TxPDO Toggle
//     Drive/Inputs/In/nState4 @bit 1 <-> WcState/InputToggle
//     Drive/Inputs/In/nState4 <-> WcState/WcState
//     Drive/Outputs/Out/nCtrl1 <-> STM Control/Control/Enable
//     Drive/Outputs/Out/nCtrl1 @bit 2 <-> STM Control/Control/Reduce torque
//     Drive/Outputs/Out/nCtrl1 @bit 1 <-> STM Control/Control/Reset
//     Drive/Outputs/Out/nDataOut2[0] <-> STM Velocity/Velocity
//     Enc/Inputs/In/nDataIn1[0] <-> ENC Status compact/Counter value
//     Enc/Inputs/In/nDataIn2[0] <-> ENC Status compact/Latch value
//     Enc/Inputs/In/nState1 @bit 4 <-> ENC Status compact/Status/Counter overflow
//     Enc/Inputs/In/nState1 @bit 3 <-> ENC Status compact/Status/Counter underflow
//     Enc/Inputs/In/nState1 @bit 1 <-> ENC Status compact/Status/Latch extern valid
//     Enc/Inputs/In/nState1 @bit 2 <-> ENC Status compact/Status/Set counter done
//     Enc/Inputs/In/nState2 @bit 4 <-> ENC Status compact/Status/Status of extern latch
//     Enc/Inputs/In/nState2 @bit 5 <-> ENC Status compact/Status/Sync error
//     Enc/Inputs/In/nState2 @bit 7 <-> ENC Status compact/Status/TxPDO Toggle
//     Enc/Inputs/In/nState4 @bit 1 <-> WcState/InputToggle
//     Enc/Inputs/In/nState4 <-> WcState/WcState
//     Enc/Outputs/Out/nCtrl1 @bit 3 <-> ENC Control compact/Control/Enable latch extern on negative edge
//     Enc/Outputs/Out/nCtrl1 @bit 1 <-> ENC Control compact/Control/Enable latch extern on positive edge
//     Enc/Outputs/Out/nCtrl1 @bit 2 <-> ENC Control compact/Control/Set counter
//     Enc/Outputs/Out/nDataOut1[0] <-> ENC Control compact/Set counter value
//   (this object) <-> Device 1 (EtherCAT)/Term 1 (EK1200)/Term 11 (EK1122)/Term 12 (EK1100)/Term 14 (EL7031)
//     Drive/Inputs/In/nState1 @bit 3 <-> STM Status/Status/Error
//     Drive/Inputs/In/nState1 @bit 5 <-> STM Status/Status/Moving negative
//     Drive/Inputs/In/nState1 @bit 4 <-> STM Status/Status/Moving positive
//     Drive/Inputs/In/nState1 @bit 1 <-> STM Status/Status/Ready
//     Drive/Inputs/In/nState1 <-> STM Status/Status/Ready to enable
//     Drive/Inputs/In/nState1 @bit 6 <-> STM Status/Status/Torque reduced
//     Drive/Inputs/In/nState1 @bit 2 <-> STM Status/Status/Warning
//     Drive/Inputs/In/nState2 @bit 3 <-> STM Status/Status/Digital input 1
//     Drive/Inputs/In/nState2 @bit 4 <-> STM Status/Status/Digital input 2
//     Drive/Inputs/In/nState2 @bit 5 <-> STM Status/Status/Sync error
//     Drive/Inputs/In/nState2 @bit 7 <-> STM Status/Status/TxPDO Toggle
//     Drive/Inputs/In/nState4 @bit 1 <-> WcState/InputToggle
//     Drive/Inputs/In/nState4 <-> WcState/WcState
//     Drive/Outputs/Out/nCtrl1 <-> STM Control/Control/Enable
//     Drive/Outputs/Out/nCtrl1 @bit 2 <-> STM Control/Control/Reduce torque
//     Drive/Outputs/Out/nCtrl1 @bit 1 <-> STM Control/Control/Reset
//     Drive/Outputs/Out/nDataOut2[0] <-> STM Velocity/Velocity
//     Enc/Inputs/In/nDataIn1[0] <-> ENC Status compact/Counter value
//     Enc/Inputs/In/nDataIn2[0] <-> ENC Status compact/Latch value
//     Enc/Inputs/In/nState1 @bit 4 <-> ENC Status compact/Status/Counter overflow
//     Enc/Inputs/In/nState1 @bit 3 <-> ENC Status compact/Status/Counter underflow
//     Enc/Inputs/In/nState1 @bit 1 <-> ENC Status compact/Status/Latch extern valid
//     Enc/Inputs/In/nState1 @bit 2 <-> ENC Status compact/Status/Set counter done
//     Enc/Inputs/In/nState2 @bit 4 <-> ENC Status compact/Status/Status of extern latch
//     Enc/Inputs/In/nState2 @bit 5 <-> ENC Status compact/Status/Sync error
//     Enc/Inputs/In/nState2 @bit 7 <-> ENC Status compact/Status/TxPDO Toggle
//     Enc/Inputs/In/nState4 @bit 1 <-> WcState/InputToggle
//     Enc/Inputs/In/nState4 <-> WcState/WcState
//     Enc/Outputs/Out/nCtrl1 @bit 3 <-> ENC Control compact/Control/Enable latch extern on negative edge
//     Enc/Outputs/Out/nCtrl1 @bit 1 <-> ENC Control compact/Control/Enable latch extern on positive edge
//     Enc/Outputs/Out/nCtrl1 @bit 2 <-> ENC Control compact/Control/Set counter
//     Enc/Outputs/Out/nDataOut1[0] <-> ENC Control compact/Set counter value
//   (this object) <-> Device 1 (EtherCAT)/Term 1 (EK1200)/Term 11 (EK1122)/Term 12 (EK1100)/Term 16 (EL7031)
//     Drive/Inputs/In/nState1 @bit 3 <-> STM Status/Status/Error
//     Drive/Inputs/In/nState1 @bit 5 <-> STM Status/Status/Moving negative
//     Drive/Inputs/In/nState1 @bit 4 <-> STM Status/Status/Moving positive
//     Drive/Inputs/In/nState1 @bit 1 <-> STM Status/Status/Ready
//     Drive/Inputs/In/nState1 <-> STM Status/Status/Ready to enable
//     Drive/Inputs/In/nState1 @bit 6 <-> STM Status/Status/Torque reduced
//     Drive/Inputs/In/nState1 @bit 2 <-> STM Status/Status/Warning
//     Drive/Inputs/In/nState2 @bit 3 <-> STM Status/Status/Digital input 1
//     Drive/Inputs/In/nState2 @bit 4 <-> STM Status/Status/Digital input 2
//     Drive/Inputs/In/nState2 @bit 5 <-> STM Status/Status/Sync error
//     Drive/Inputs/In/nState2 @bit 7 <-> STM Status/Status/TxPDO Toggle
//     Drive/Inputs/In/nState4 @bit 1 <-> WcState/InputToggle
//     Drive/Inputs/In/nState4 <-> WcState/WcState
//     Drive/Outputs/Out/nCtrl1 <-> STM Control/Control/Enable
//     Drive/Outputs/Out/nCtrl1 @bit 2 <-> STM Control/Control/Reduce torque
//     Drive/Outputs/Out/nCtrl1 @bit 1 <-> STM Control/Control/Reset
//     Drive/Outputs/Out/nDataOut2[0] <-> STM Velocity/Velocity
//     Enc/Inputs/In/nDataIn1[0] <-> ENC Status compact/Counter value
//     Enc/Inputs/In/nDataIn2[0] <-> ENC Status compact/Latch value
//     Enc/Inputs/In/nState1 @bit 4 <-> ENC Status compact/Status/Counter overflow
//     Enc/Inputs/In/nState1 @bit 3 <-> ENC Status compact/Status/Counter underflow
//     Enc/Inputs/In/nState1 @bit 1 <-> ENC Status compact/Status/Latch extern valid
//     Enc/Inputs/In/nState1 @bit 2 <-> ENC Status compact/Status/Set counter done
//     Enc/Inputs/In/nState2 @bit 4 <-> ENC Status compact/Status/Status of extern latch
//     Enc/Inputs/In/nState2 @bit 5 <-> ENC Status compact/Status/Sync error
//     Enc/Inputs/In/nState2 @bit 7 <-> ENC Status compact/Status/TxPDO Toggle
//     Enc/Inputs/In/nState4 @bit 1 <-> WcState/InputToggle
//     Enc/Inputs/In/nState4 <-> WcState/WcState
//     Enc/Outputs/Out/nCtrl1 @bit 3 <-> ENC Control compact/Control/Enable latch extern on negative edge
//     Enc/Outputs/Out/nCtrl1 @bit 1 <-> ENC Control compact/Control/Enable latch extern on positive edge
//     Enc/Outputs/Out/nCtrl1 @bit 2 <-> ENC Control compact/Control/Set counter
//     Enc/Outputs/Out/nDataOut1[0] <-> ENC Control compact/Set counter value
//   (this object) <-> Device 1 (EtherCAT)/Term 1 (EK1200)/Term 11 (EK1122)/Term 12 (EK1100)/Term 17 (EL7031)
//     Drive/Inputs/In/nState1 @bit 3 <-> STM Status/Status/Error
//     Drive/Inputs/In/nState1 @bit 5 <-> STM Status/Status/Moving negative
//     Drive/Inputs/In/nState1 @bit 4 <-> STM Status/Status/Moving positive
//     Drive/Inputs/In/nState1 @bit 1 <-> STM Status/Status/Ready
//     Drive/Inputs/In/nState1 <-> STM Status/Status/Ready to enable
//     Drive/Inputs/In/nState1 @bit 6 <-> STM Status/Status/Torque reduced
//     Drive/Inputs/In/nState1 @bit 2 <-> STM Status/Status/Warning
//     Drive/Inputs/In/nState2 @bit 3 <-> STM Status/Status/Digital input 1
//     Drive/Inputs/In/nState2 @bit 4 <-> STM Status/Status/Digital input 2
//     Drive/Inputs/In/nState2 @bit 5 <-> STM Status/Status/Sync error
//     Drive/Inputs/In/nState2 @bit 7 <-> STM Status/Status/TxPDO Toggle
//     Drive/Inputs/In/nState4 @bit 1 <-> WcState/InputToggle
//     Drive/Inputs/In/nState4 <-> WcState/WcState
//     Drive/Outputs/Out/nCtrl1 <-> STM Control/Control/Enable
//     Drive/Outputs/Out/nCtrl1 @bit 2 <-> STM Control/Control/Reduce torque
//     Drive/Outputs/Out/nCtrl1 @bit 1 <-> STM Control/Control/Reset
//     Drive/Outputs/Out/nDataOut2[0] <-> STM Velocity/Velocity
//     Enc/Inputs/In/nDataIn1[0] <-> ENC Status compact/Counter value
//     Enc/Inputs/In/nDataIn2[0] <-> ENC Status compact/Latch value
//     Enc/Inputs/In/nState1 @bit 4 <-> ENC Status compact/Status/Counter overflow
//     Enc/Inputs/In/nState1 @bit 3 <-> ENC Status compact/Status/Counter underflow
//     Enc/Inputs/In/nState1 @bit 1 <-> ENC Status compact/Status/Latch extern valid
//     Enc/Inputs/In/nState1 @bit 2 <-> ENC Status compact/Status/Set counter done
//     Enc/Inputs/In/nState2 @bit 4 <-> ENC Status compact/Status/Status of extern latch
//     Enc/Inputs/In/nState2 @bit 5 <-> ENC Status compact/Status/Sync error
//     Enc/Inputs/In/nState2 @bit 7 <-> ENC Status compact/Status/TxPDO Toggle
//     Enc/Inputs/In/nState4 @bit 1 <-> WcState/InputToggle
//     Enc/Inputs/In/nState4 <-> WcState/WcState
//     Enc/Outputs/Out/nCtrl1 @bit 3 <-> ENC Control compact/Control/Enable latch extern on negative edge
//     Enc/Outputs/Out/nCtrl1 @bit 1 <-> ENC Control compact/Control/Enable latch extern on positive edge
//     Enc/Outputs/Out/nCtrl1 @bit 2 <-> ENC Control compact/Control/Set counter
//     Enc/Outputs/Out/nDataOut1[0] <-> ENC Control compact/Set counter value
//   (this object) <-> Device 1 (EtherCAT)/Term 1 (EK1200)/Term 11 (EK1122)/Term 12 (EK1100)/Term 18 (EL7031)
//     Drive/Inputs/In/nState1 @bit 3 <-> STM Status/Status/Error
//     Drive/Inputs/In/nState1 @bit 5 <-> STM Status/Status/Moving negative
//     Drive/Inputs/In/nState1 @bit 4 <-> STM Status/Status/Moving positive
//     Drive/Inputs/In/nState1 @bit 1 <-> STM Status/Status/Ready
//     Drive/Inputs/In/nState1 <-> STM Status/Status/Ready to enable
//     Drive/Inputs/In/nState1 @bit 6 <-> STM Status/Status/Torque reduced
//     Drive/Inputs/In/nState1 @bit 2 <-> STM Status/Status/Warning
//     Drive/Inputs/In/nState2 @bit 3 <-> STM Status/Status/Digital input 1
//     Drive/Inputs/In/nState2 @bit 4 <-> STM Status/Status/Digital input 2
//     Drive/Inputs/In/nState2 @bit 5 <-> STM Status/Status/Sync error
//     Drive/Inputs/In/nState2 @bit 7 <-> STM Status/Status/TxPDO Toggle
//     Drive/Inputs/In/nState4 @bit 1 <-> WcState/InputToggle
//     Drive/Inputs/In/nState4 <-> WcState/WcState
//     Drive/Outputs/Out/nCtrl1 <-> STM Control/Control/Enable
//     Drive/Outputs/Out/nCtrl1 @bit 2 <-> STM Control/Control/Reduce torque
//     Drive/Outputs/Out/nCtrl1 @bit 1 <-> STM Control/Control/Reset
//     Drive/Outputs/Out/nDataOut2[0] <-> STM Velocity/Velocity
//     Enc/Inputs/In/nDataIn1[0] <-> ENC Status compact/Counter value
//     Enc/Inputs/In/nDataIn2[0] <-> ENC Status compact/Latch value
//     Enc/Inputs/In/nState1 @bit 4 <-> ENC Status compact/Status/Counter overflow
//     Enc/Inputs/In/nState1 @bit 3 <-> ENC Status compact/Status/Counter underflow
//     Enc/Inputs/In/nState1 @bit 1 <-> ENC Status compact/Status/Latch extern valid
//     Enc/Inputs/In/nState1 @bit 2 <-> ENC Status compact/Status/Set counter done
//     Enc/Inputs/In/nState2 @bit 4 <-> ENC Status compact/Status/Status of extern latch
//     Enc/Inputs/In/nState2 @bit 5 <-> ENC Status compact/Status/Sync error
//     Enc/Inputs/In/nState2 @bit 7 <-> ENC Status compact/Status/TxPDO Toggle
//     Enc/Inputs/In/nState4 @bit 1 <-> WcState/InputToggle
//     Enc/Inputs/In/nState4 <-> WcState/WcState
//     Enc/Outputs/Out/nCtrl1 @bit 3 <-> ENC Control compact/Control/Enable latch extern on negative edge
//     Enc/Outputs/Out/nCtrl1 @bit 1 <-> ENC Control compact/Control/Enable latch extern on positive edge
//     Enc/Outputs/Out/nCtrl1 @bit 2 <-> ENC Control compact/Control/Set counter
//     Enc/Outputs/Out/nDataOut1[0] <-> ENC Control compact/Set counter value
//   (this object) <-> Device 1 (EtherCAT)/Term 1 (EK1200)/Term 11 (EK1122)/Term 12 (EK1100)/Term 19 (EL7031)
//     Drive/Inputs/In/nState1 @bit 3 <-> STM Status/Status/Error
//     Drive/Inputs/In/nState1 @bit 5 <-> STM Status/Status/Moving negative
//     Drive/Inputs/In/nState1 @bit 4 <-> STM Status/Status/Moving positive
//     Drive/Inputs/In/nState1 @bit 1 <-> STM Status/Status/Ready
//     Drive/Inputs/In/nState1 <-> STM Status/Status/Ready to enable
//     Drive/Inputs/In/nState1 @bit 6 <-> STM Status/Status/Torque reduced
//     Drive/Inputs/In/nState1 @bit 2 <-> STM Status/Status/Warning
//     Drive/Inputs/In/nState2 @bit 3 <-> STM Status/Status/Digital input 1
//     Drive/Inputs/In/nState2 @bit 4 <-> STM Status/Status/Digital input 2
//     Drive/Inputs/In/nState2 @bit 5 <-> STM Status/Status/Sync error
//     Drive/Inputs/In/nState2 @bit 7 <-> STM Status/Status/TxPDO Toggle
//     Drive/Inputs/In/nState4 @bit 1 <-> WcState/InputToggle
//     Drive/Inputs/In/nState4 <-> WcState/WcState
//     Drive/Outputs/Out/nCtrl1 <-> STM Control/Control/Enable
//     Drive/Outputs/Out/nCtrl1 @bit 2 <-> STM Control/Control/Reduce torque
//     Drive/Outputs/Out/nCtrl1 @bit 1 <-> STM Control/Control/Reset
//     Drive/Outputs/Out/nDataOut2[0] <-> STM Velocity/Velocity
//     Enc/Inputs/In/nDataIn1[0] <-> ENC Status compact/Counter value
//     Enc/Inputs/In/nDataIn2[0] <-> ENC Status compact/Latch value
//     Enc/Inputs/In/nState1 @bit 4 <-> ENC Status compact/Status/Counter overflow
//     Enc/Inputs/In/nState1 @bit 3 <-> ENC Status compact/Status/Counter underflow
//     Enc/Inputs/In/nState1 @bit 1 <-> ENC Status compact/Status/Latch extern valid
//     Enc/Inputs/In/nState1 @bit 2 <-> ENC Status compact/Status/Set counter done
//     Enc/Inputs/In/nState2 @bit 4 <-> ENC Status compact/Status/Status of extern latch
//     Enc/Inputs/In/nState2 @bit 5 <-> ENC Status compact/Status/Sync error
//     Enc/Inputs/In/nState2 @bit 7 <-> ENC Status compact/Status/TxPDO Toggle
//     Enc/Inputs/In/nState4 @bit 1 <-> WcState/InputToggle
//     Enc/Inputs/In/nState4 <-> WcState/WcState
//     Enc/Outputs/Out/nCtrl1 @bit 3 <-> ENC Control compact/Control/Enable latch extern on negative edge
//     Enc/Outputs/Out/nCtrl1 @bit 1 <-> ENC Control compact/Control/Enable latch extern on positive edge
//     Enc/Outputs/Out/nCtrl1 @bit 2 <-> ENC Control compact/Control/Set counter
//     Enc/Outputs/Out/nDataOut1[0] <-> ENC Control compact/Set counter value
//   (this object) <-> Device 1 (EtherCAT)/Term 1 (EK1200)/Term 11 (EK1122)/Term 12 (EK1100)/Term 21 (EL7031)
//     Drive/Inputs/In/nState1 @bit 3 <-> STM Status/Status/Error
//     Drive/Inputs/In/nState1 @bit 5 <-> STM Status/Status/Moving negative
//     Drive/Inputs/In/nState1 @bit 4 <-> STM Status/Status/Moving positive
//     Drive/Inputs/In/nState1 @bit 1 <-> STM Status/Status/Ready
//     Drive/Inputs/In/nState1 <-> STM Status/Status/Ready to enable
//     Drive/Inputs/In/nState1 @bit 6 <-> STM Status/Status/Torque reduced
//     Drive/Inputs/In/nState1 @bit 2 <-> STM Status/Status/Warning
//     Drive/Inputs/In/nState2 @bit 3 <-> STM Status/Status/Digital input 1
//     Drive/Inputs/In/nState2 @bit 4 <-> STM Status/Status/Digital input 2
//     Drive/Inputs/In/nState2 @bit 5 <-> STM Status/Status/Sync error
//     Drive/Inputs/In/nState2 @bit 7 <-> STM Status/Status/TxPDO Toggle
//     Drive/Inputs/In/nState4 @bit 1 <-> WcState/InputToggle
//     Drive/Inputs/In/nState4 <-> WcState/WcState
//     Drive/Outputs/Out/nCtrl1 <-> STM Control/Control/Enable
//     Drive/Outputs/Out/nCtrl1 @bit 2 <-> STM Control/Control/Reduce torque
//     Drive/Outputs/Out/nCtrl1 @bit 1 <-> STM Control/Control/Reset
//     Drive/Outputs/Out/nDataOut2[0] <-> STM Velocity/Velocity
//     Enc/Inputs/In/nDataIn1[0] <-> ENC Status compact/Counter value
//     Enc/Inputs/In/nDataIn2[0] <-> ENC Status compact/Latch value
//     Enc/Inputs/In/nState1 @bit 4 <-> ENC Status compact/Status/Counter overflow
//     Enc/Inputs/In/nState1 @bit 3 <-> ENC Status compact/Status/Counter underflow
//     Enc/Inputs/In/nState1 @bit 1 <-> ENC Status compact/Status/Latch extern valid
//     Enc/Inputs/In/nState1 @bit 2 <-> ENC Status compact/Status/Set counter done
//     Enc/Inputs/In/nState2 @bit 4 <-> ENC Status compact/Status/Status of extern latch
//     Enc/Inputs/In/nState2 @bit 5 <-> ENC Status compact/Status/Sync error
//     Enc/Inputs/In/nState2 @bit 7 <-> ENC Status compact/Status/TxPDO Toggle
//     Enc/Inputs/In/nState4 @bit 1 <-> WcState/InputToggle
//     Enc/Inputs/In/nState4 <-> WcState/WcState
//     Enc/Outputs/Out/nCtrl1 @bit 3 <-> ENC Control compact/Control/Enable latch extern on negative edge
//     Enc/Outputs/Out/nCtrl1 @bit 1 <-> ENC Control compact/Control/Enable latch extern on positive edge
//     Enc/Outputs/Out/nCtrl1 @bit 2 <-> ENC Control compact/Control/Set counter
//     Enc/Outputs/Out/nDataOut1[0] <-> ENC Control compact/Set counter value
//   (this object) <-> Device 1 (EtherCAT)/Term 1 (EK1200)/Term 11 (EK1122)/Term 12 (EK1100)/Term 22 (EL7031)
//     Drive/Inputs/In/nState1 @bit 3 <-> STM Status/Status/Error
//     Drive/Inputs/In/nState1 @bit 5 <-> STM Status/Status/Moving negative
//     Drive/Inputs/In/nState1 @bit 4 <-> STM Status/Status/Moving positive
//     Drive/Inputs/In/nState1 @bit 1 <-> STM Status/Status/Ready
//     Drive/Inputs/In/nState1 <-> STM Status/Status/Ready to enable
//     Drive/Inputs/In/nState1 @bit 6 <-> STM Status/Status/Torque reduced
//     Drive/Inputs/In/nState1 @bit 2 <-> STM Status/Status/Warning
//     Drive/Inputs/In/nState2 @bit 3 <-> STM Status/Status/Digital input 1
//     Drive/Inputs/In/nState2 @bit 4 <-> STM Status/Status/Digital input 2
//     Drive/Inputs/In/nState2 @bit 5 <-> STM Status/Status/Sync error
//     Drive/Inputs/In/nState2 @bit 7 <-> STM Status/Status/TxPDO Toggle
//     Drive/Inputs/In/nState4 @bit 1 <-> WcState/InputToggle
//     Drive/Inputs/In/nState4 <-> WcState/WcState
//     Drive/Outputs/Out/nCtrl1 <-> STM Control/Control/Enable
//     Drive/Outputs/Out/nCtrl1 @bit 2 <-> STM Control/Control/Reduce torque
//     Drive/Outputs/Out/nCtrl1 @bit 1 <-> STM Control/Control/Reset
//     Drive/Outputs/Out/nDataOut2[0] <-> STM Velocity/Velocity
//     Enc/Inputs/In/nDataIn1[0] <-> ENC Status compact/Counter value
//     Enc/Inputs/In/nDataIn2[0] <-> ENC Status compact/Latch value
//     Enc/Inputs/In/nState1 @bit 4 <-> ENC Status compact/Status/Counter overflow
//     Enc/Inputs/In/nState1 @bit 3 <-> ENC Status compact/Status/Counter underflow
//     Enc/Inputs/In/nState1 @bit 1 <-> ENC Status compact/Status/Latch extern valid
//     Enc/Inputs/In/nState1 @bit 2 <-> ENC Status compact/Status/Set counter done
//     Enc/Inputs/In/nState2 @bit 4 <-> ENC Status compact/Status/Status of extern latch
//     Enc/Inputs/In/nState2 @bit 5 <-> ENC Status compact/Status/Sync error
//     Enc/Inputs/In/nState2 @bit 7 <-> ENC Status compact/Status/TxPDO Toggle
//     Enc/Inputs/In/nState4 @bit 1 <-> WcState/InputToggle
//     Enc/Inputs/In/nState4 <-> WcState/WcState
//     Enc/Outputs/Out/nCtrl1 @bit 3 <-> ENC Control compact/Control/Enable latch extern on negative edge
//     Enc/Outputs/Out/nCtrl1 @bit 1 <-> ENC Control compact/Control/Enable latch extern on positive edge
//     Enc/Outputs/Out/nCtrl1 @bit 2 <-> ENC Control compact/Control/Set counter
//     Enc/Outputs/Out/nDataOut1[0] <-> ENC Control compact/Set counter value
//   (this object) <-> Device 1 (EtherCAT)/Term 1 (EK1200)/Term 11 (EK1122)/Term 12 (EK1100)/Term 24 (EL7031)
//     Drive/Inputs/In/nState1 @bit 3 <-> STM Status/Status/Error
//     Drive/Inputs/In/nState1 @bit 5 <-> STM Status/Status/Moving negative
//     Drive/Inputs/In/nState1 @bit 4 <-> STM Status/Status/Moving positive
//     Drive/Inputs/In/nState1 @bit 1 <-> STM Status/Status/Ready
//     Drive/Inputs/In/nState1 <-> STM Status/Status/Ready to enable
//     Drive/Inputs/In/nState1 @bit 6 <-> STM Status/Status/Torque reduced
//     Drive/Inputs/In/nState1 @bit 2 <-> STM Status/Status/Warning
//     Drive/Inputs/In/nState2 @bit 3 <-> STM Status/Status/Digital input 1
//     Drive/Inputs/In/nState2 @bit 4 <-> STM Status/Status/Digital input 2
//     Drive/Inputs/In/nState2 @bit 5 <-> STM Status/Status/Sync error
//     Drive/Inputs/In/nState2 @bit 7 <-> STM Status/Status/TxPDO Toggle
//     Drive/Inputs/In/nState4 @bit 1 <-> WcState/InputToggle
//     Drive/Inputs/In/nState4 <-> WcState/WcState
//     Drive/Outputs/Out/nCtrl1 <-> STM Control/Control/Enable
//     Drive/Outputs/Out/nCtrl1 @bit 2 <-> STM Control/Control/Reduce torque
//     Drive/Outputs/Out/nCtrl1 @bit 1 <-> STM Control/Control/Reset
//     Drive/Outputs/Out/nDataOut2[0] <-> STM Velocity/Velocity
//     Enc/Inputs/In/nDataIn1[0] <-> ENC Status compact/Counter value
//     Enc/Inputs/In/nDataIn2[0] <-> ENC Status compact/Latch value
//     Enc/Inputs/In/nState1 @bit 4 <-> ENC Status compact/Status/Counter overflow
//     Enc/Inputs/In/nState1 @bit 3 <-> ENC Status compact/Status/Counter underflow
//     Enc/Inputs/In/nState1 @bit 1 <-> ENC Status compact/Status/Latch extern valid
//     Enc/Inputs/In/nState1 @bit 2 <-> ENC Status compact/Status/Set counter done
//     Enc/Inputs/In/nState2 @bit 4 <-> ENC Status compact/Status/Status of extern latch
//     Enc/Inputs/In/nState2 @bit 5 <-> ENC Status compact/Status/Sync error
//     Enc/Inputs/In/nState2 @bit 7 <-> ENC Status compact/Status/TxPDO Toggle
//     Enc/Inputs/In/nState4 @bit 1 <-> WcState/InputToggle
//     Enc/Inputs/In/nState4 <-> WcState/WcState
//     Enc/Outputs/Out/nCtrl1 @bit 3 <-> ENC Control compact/Control/Enable latch extern on negative edge
//     Enc/Outputs/Out/nCtrl1 @bit 1 <-> ENC Control compact/Control/Enable latch extern on positive edge
//     Enc/Outputs/Out/nCtrl1 @bit 2 <-> ENC Control compact/Control/Set counter
//     Enc/Outputs/Out/nDataOut1[0] <-> ENC Control compact/Set counter value
//   (this object) <-> Device 1 (EtherCAT)/Term 1 (EK1200)/Term 11 (EK1122)/Term 12 (EK1100)/Term 25 (EL7031)
//     Drive/Inputs/In/nState1 @bit 3 <-> STM Status/Status/Error
//     Drive/Inputs/In/nState1 @bit 5 <-> STM Status/Status/Moving negative
//     Drive/Inputs/In/nState1 @bit 4 <-> STM Status/Status/Moving positive
//     Drive/Inputs/In/nState1 @bit 1 <-> STM Status/Status/Ready
//     Drive/Inputs/In/nState1 <-> STM Status/Status/Ready to enable
//     Drive/Inputs/In/nState1 @bit 6 <-> STM Status/Status/Torque reduced
//     Drive/Inputs/In/nState1 @bit 2 <-> STM Status/Status/Warning
//     Drive/Inputs/In/nState2 @bit 3 <-> STM Status/Status/Digital input 1
//     Drive/Inputs/In/nState2 @bit 4 <-> STM Status/Status/Digital input 2
//     Drive/Inputs/In/nState2 @bit 5 <-> STM Status/Status/Sync error
//     Drive/Inputs/In/nState2 @bit 7 <-> STM Status/Status/TxPDO Toggle
//     Drive/Inputs/In/nState4 @bit 1 <-> WcState/InputToggle
//     Drive/Inputs/In/nState4 <-> WcState/WcState
//     Drive/Outputs/Out/nCtrl1 <-> STM Control/Control/Enable
//     Drive/Outputs/Out/nCtrl1 @bit 2 <-> STM Control/Control/Reduce torque
//     Drive/Outputs/Out/nCtrl1 @bit 1 <-> STM Control/Control/Reset
//     Drive/Outputs/Out/nDataOut2[0] <-> STM Velocity/Velocity
//     Enc/Inputs/In/nDataIn1[0] <-> ENC Status compact/Counter value
//     Enc/Inputs/In/nDataIn2[0] <-> ENC Status compact/Latch value
//     Enc/Inputs/In/nState1 @bit 4 <-> ENC Status compact/Status/Counter overflow
//     Enc/Inputs/In/nState1 @bit 3 <-> ENC Status compact/Status/Counter underflow
//     Enc/Inputs/In/nState1 @bit 1 <-> ENC Status compact/Status/Latch extern valid
//     Enc/Inputs/In/nState1 @bit 2 <-> ENC Status compact/Status/Set counter done
//     Enc/Inputs/In/nState2 @bit 4 <-> ENC Status compact/Status/Status of extern latch
//     Enc/Inputs/In/nState2 @bit 5 <-> ENC Status compact/Status/Sync error
//     Enc/Inputs/In/nState2 @bit 7 <-> ENC Status compact/Status/TxPDO Toggle
//     Enc/Inputs/In/nState4 @bit 1 <-> WcState/InputToggle
//     Enc/Inputs/In/nState4 <-> WcState/WcState
//     Enc/Outputs/Out/nCtrl1 @bit 3 <-> ENC Control compact/Control/Enable latch extern on negative edge
//     Enc/Outputs/Out/nCtrl1 @bit 1 <-> ENC Control compact/Control/Enable latch extern on positive edge
//     Enc/Outputs/Out/nCtrl1 @bit 2 <-> ENC Control compact/Control/Set counter
//     Enc/Outputs/Out/nDataOut1[0] <-> ENC Control compact/Set counter value
//   (this object) <-> Device 1 (EtherCAT)/Term 1 (EK1200)/Term 11 (EK1122)/Term 12 (EK1100)/Term 27 (EL7031)
//     Drive/Inputs/In/nState1 @bit 3 <-> STM Status/Status/Error
//     Drive/Inputs/In/nState1 @bit 5 <-> STM Status/Status/Moving negative
//     Drive/Inputs/In/nState1 @bit 4 <-> STM Status/Status/Moving positive
//     Drive/Inputs/In/nState1 @bit 1 <-> STM Status/Status/Ready
//     Drive/Inputs/In/nState1 <-> STM Status/Status/Ready to enable
//     Drive/Inputs/In/nState1 @bit 6 <-> STM Status/Status/Torque reduced
//     Drive/Inputs/In/nState1 @bit 2 <-> STM Status/Status/Warning
//     Drive/Inputs/In/nState2 @bit 3 <-> STM Status/Status/Digital input 1
//     Drive/Inputs/In/nState2 @bit 4 <-> STM Status/Status/Digital input 2
//     Drive/Inputs/In/nState2 @bit 5 <-> STM Status/Status/Sync error
//     Drive/Inputs/In/nState2 @bit 7 <-> STM Status/Status/TxPDO Toggle
//     Drive/Inputs/In/nState4 @bit 1 <-> WcState/InputToggle
//     Drive/Inputs/In/nState4 <-> WcState/WcState
//     Drive/Outputs/Out/nCtrl1 <-> STM Control/Control/Enable
//     Drive/Outputs/Out/nCtrl1 @bit 2 <-> STM Control/Control/Reduce torque
//     Drive/Outputs/Out/nCtrl1 @bit 1 <-> STM Control/Control/Reset
//     Drive/Outputs/Out/nDataOut2[0] <-> STM Velocity/Velocity
//     Enc/Inputs/In/nDataIn1[0] <-> ENC Status compact/Counter value
//     Enc/Inputs/In/nDataIn2[0] <-> ENC Status compact/Latch value
//     Enc/Inputs/In/nState1 @bit 4 <-> ENC Status compact/Status/Counter overflow
//     Enc/Inputs/In/nState1 @bit 3 <-> ENC Status compact/Status/Counter underflow
//     Enc/Inputs/In/nState1 @bit 1 <-> ENC Status compact/Status/Latch extern valid
//     Enc/Inputs/In/nState1 @bit 2 <-> ENC Status compact/Status/Set counter done
//     Enc/Inputs/In/nState2 @bit 4 <-> ENC Status compact/Status/Status of extern latch
//     Enc/Inputs/In/nState2 @bit 5 <-> ENC Status compact/Status/Sync error
//     Enc/Inputs/In/nState2 @bit 7 <-> ENC Status compact/Status/TxPDO Toggle
//     Enc/Inputs/In/nState4 @bit 1 <-> WcState/InputToggle
//     Enc/Inputs/In/nState4 <-> WcState/WcState
//     Enc/Outputs/Out/nCtrl1 @bit 3 <-> ENC Control compact/Control/Enable latch extern on negative edge
//     Enc/Outputs/Out/nCtrl1 @bit 1 <-> ENC Control compact/Control/Enable latch extern on positive edge
//     Enc/Outputs/Out/nCtrl1 @bit 2 <-> ENC Control compact/Control/Set counter
//     Enc/Outputs/Out/nDataOut1[0] <-> ENC Control compact/Set counter value
//   (this object) <-> Device 1 (EtherCAT)/Term 1 (EK1200)/Term 11 (EK1122)/Term 12 (EK1100)/Term 28 (EL7031)
//     Drive/Inputs/In/nState1 @bit 3 <-> STM Status/Status/Error
//     Drive/Inputs/In/nState1 @bit 5 <-> STM Status/Status/Moving negative
//     Drive/Inputs/In/nState1 @bit 4 <-> STM Status/Status/Moving positive
//     Drive/Inputs/In/nState1 @bit 1 <-> STM Status/Status/Ready
//     Drive/Inputs/In/nState1 <-> STM Status/Status/Ready to enable
//     Drive/Inputs/In/nState1 @bit 6 <-> STM Status/Status/Torque reduced
//     Drive/Inputs/In/nState1 @bit 2 <-> STM Status/Status/Warning
//     Drive/Inputs/In/nState2 @bit 3 <-> STM Status/Status/Digital input 1
//     Drive/Inputs/In/nState2 @bit 4 <-> STM Status/Status/Digital input 2
//     Drive/Inputs/In/nState2 @bit 5 <-> STM Status/Status/Sync error
//     Drive/Inputs/In/nState2 @bit 7 <-> STM Status/Status/TxPDO Toggle
//     Drive/Inputs/In/nState4 @bit 1 <-> WcState/InputToggle
//     Drive/Inputs/In/nState4 <-> WcState/WcState
//     Drive/Outputs/Out/nCtrl1 <-> STM Control/Control/Enable
//     Drive/Outputs/Out/nCtrl1 @bit 2 <-> STM Control/Control/Reduce torque
//     Drive/Outputs/Out/nCtrl1 @bit 1 <-> STM Control/Control/Reset
//     Drive/Outputs/Out/nDataOut2[0] <-> STM Velocity/Velocity
//     Enc/Inputs/In/nDataIn1[0] <-> ENC Status compact/Counter value
//     Enc/Inputs/In/nDataIn2[0] <-> ENC Status compact/Latch value
//     Enc/Inputs/In/nState1 @bit 4 <-> ENC Status compact/Status/Counter overflow
//     Enc/Inputs/In/nState1 @bit 3 <-> ENC Status compact/Status/Counter underflow
//     Enc/Inputs/In/nState1 @bit 1 <-> ENC Status compact/Status/Latch extern valid
//     Enc/Inputs/In/nState1 @bit 2 <-> ENC Status compact/Status/Set counter done
//     Enc/Inputs/In/nState2 @bit 4 <-> ENC Status compact/Status/Status of extern latch
//     Enc/Inputs/In/nState2 @bit 5 <-> ENC Status compact/Status/Sync error
//     Enc/Inputs/In/nState2 @bit 7 <-> ENC Status compact/Status/TxPDO Toggle
//     Enc/Inputs/In/nState4 @bit 1 <-> WcState/InputToggle
//     Enc/Inputs/In/nState4 <-> WcState/WcState
//     Enc/Outputs/Out/nCtrl1 @bit 3 <-> ENC Control compact/Control/Enable latch extern on negative edge
//     Enc/Outputs/Out/nCtrl1 @bit 1 <-> ENC Control compact/Control/Enable latch extern on positive edge
//     Enc/Outputs/Out/nCtrl1 @bit 2 <-> ENC Control compact/Control/Set counter
//     Enc/Outputs/Out/nDataOut1[0] <-> ENC Control compact/Set counter value
//   (this object) <-> Device 1 (EtherCAT)/Term 1 (EK1200)/Term 11 (EK1122)/Term 12 (EK1100)/Term 29 (EL7031)
//     Drive/Inputs/In/nState1 @bit 3 <-> STM Status/Status/Error
//     Drive/Inputs/In/nState1 @bit 5 <-> STM Status/Status/Moving negative
//     Drive/Inputs/In/nState1 @bit 4 <-> STM Status/Status/Moving positive
//     Drive/Inputs/In/nState1 @bit 1 <-> STM Status/Status/Ready
//     Drive/Inputs/In/nState1 <-> STM Status/Status/Ready to enable
//     Drive/Inputs/In/nState1 @bit 6 <-> STM Status/Status/Torque reduced
//     Drive/Inputs/In/nState1 @bit 2 <-> STM Status/Status/Warning
//     Drive/Inputs/In/nState2 @bit 3 <-> STM Status/Status/Digital input 1
//     Drive/Inputs/In/nState2 @bit 4 <-> STM Status/Status/Digital input 2
//     Drive/Inputs/In/nState2 @bit 5 <-> STM Status/Status/Sync error
//     Drive/Inputs/In/nState2 @bit 7 <-> STM Status/Status/TxPDO Toggle
//     Drive/Inputs/In/nState4 @bit 1 <-> WcState/InputToggle
//     Drive/Inputs/In/nState4 <-> WcState/WcState
//     Drive/Outputs/Out/nCtrl1 <-> STM Control/Control/Enable
//     Drive/Outputs/Out/nCtrl1 @bit 2 <-> STM Control/Control/Reduce torque
//     Drive/Outputs/Out/nCtrl1 @bit 1 <-> STM Control/Control/Reset
//     Drive/Outputs/Out/nDataOut2[0] <-> STM Velocity/Velocity
//     Enc/Inputs/In/nDataIn1[0] <-> ENC Status compact/Counter value
//     Enc/Inputs/In/nDataIn2[0] <-> ENC Status compact/Latch value
//     Enc/Inputs/In/nState1 @bit 4 <-> ENC Status compact/Status/Counter overflow
//     Enc/Inputs/In/nState1 @bit 3 <-> ENC Status compact/Status/Counter underflow
//     Enc/Inputs/In/nState1 @bit 1 <-> ENC Status compact/Status/Latch extern valid
//     Enc/Inputs/In/nState1 @bit 2 <-> ENC Status compact/Status/Set counter done
//     Enc/Inputs/In/nState2 @bit 4 <-> ENC Status compact/Status/Status of extern latch
//     Enc/Inputs/In/nState2 @bit 5 <-> ENC Status compact/Status/Sync error
//     Enc/Inputs/In/nState2 @bit 7 <-> ENC Status compact/Status/TxPDO Toggle
//     Enc/Inputs/In/nState4 @bit 1 <-> WcState/InputToggle
//     Enc/Inputs/In/nState4 <-> WcState/WcState
//     Enc/Outputs/Out/nCtrl1 @bit 3 <-> ENC Control compact/Control/Enable latch extern on negative edge
//     Enc/Outputs/Out/nCtrl1 @bit 1 <-> ENC Control compact/Control/Enable latch extern on positive edge
//     Enc/Outputs/Out/nCtrl1 @bit 2 <-> ENC Control compact/Control/Set counter
//     Enc/Outputs/Out/nDataOut1[0] <-> ENC Control compact/Set counter value
//   (this object) <-> Device 1 (EtherCAT)/Term 1 (EK1200)/Term 11 (EK1122)/Term 12 (EK1100)/Term 30 (EL7031)
//     Drive/Inputs/In/nState1 @bit 3 <-> STM Status/Status/Error
//     Drive/Inputs/In/nState1 @bit 5 <-> STM Status/Status/Moving negative
//     Drive/Inputs/In/nState1 @bit 4 <-> STM Status/Status/Moving positive
//     Drive/Inputs/In/nState1 @bit 1 <-> STM Status/Status/Ready
//     Drive/Inputs/In/nState1 <-> STM Status/Status/Ready to enable
//     Drive/Inputs/In/nState1 @bit 6 <-> STM Status/Status/Torque reduced
//     Drive/Inputs/In/nState1 @bit 2 <-> STM Status/Status/Warning
//     Drive/Inputs/In/nState2 @bit 3 <-> STM Status/Status/Digital input 1
//     Drive/Inputs/In/nState2 @bit 4 <-> STM Status/Status/Digital input 2
//     Drive/Inputs/In/nState2 @bit 5 <-> STM Status/Status/Sync error
//     Drive/Inputs/In/nState2 @bit 7 <-> STM Status/Status/TxPDO Toggle
//     Drive/Inputs/In/nState4 @bit 1 <-> WcState/InputToggle
//     Drive/Inputs/In/nState4 <-> WcState/WcState
//     Drive/Outputs/Out/nCtrl1 <-> STM Control/Control/Enable
//     Drive/Outputs/Out/nCtrl1 @bit 2 <-> STM Control/Control/Reduce torque
//     Drive/Outputs/Out/nCtrl1 @bit 1 <-> STM Control/Control/Reset
//     Drive/Outputs/Out/nDataOut2[0] <-> STM Velocity/Velocity
//     Enc/Inputs/In/nDataIn1[0] <-> ENC Status compact/Counter value
//     Enc/Inputs/In/nDataIn2[0] <-> ENC Status compact/Latch value
//     Enc/Inputs/In/nState1 @bit 4 <-> ENC Status compact/Status/Counter overflow
//     Enc/Inputs/In/nState1 @bit 3 <-> ENC Status compact/Status/Counter underflow
//     Enc/Inputs/In/nState1 @bit 1 <-> ENC Status compact/Status/Latch extern valid
//     Enc/Inputs/In/nState1 @bit 2 <-> ENC Status compact/Status/Set counter done
//     Enc/Inputs/In/nState2 @bit 4 <-> ENC Status compact/Status/Status of extern latch
//     Enc/Inputs/In/nState2 @bit 5 <-> ENC Status compact/Status/Sync error
//     Enc/Inputs/In/nState2 @bit 7 <-> ENC Status compact/Status/TxPDO Toggle
//     Enc/Inputs/In/nState4 @bit 1 <-> WcState/InputToggle
//     Enc/Inputs/In/nState4 <-> WcState/WcState
//     Enc/Outputs/Out/nCtrl1 @bit 3 <-> ENC Control compact/Control/Enable latch extern on negative edge
//     Enc/Outputs/Out/nCtrl1 @bit 1 <-> ENC Control compact/Control/Enable latch extern on positive edge
//     Enc/Outputs/Out/nCtrl1 @bit 2 <-> ENC Control compact/Control/Set counter
//     Enc/Outputs/Out/nDataOut1[0] <-> ENC Control compact/Set counter value
//   (this object) <-> Device 1 (EtherCAT)/Term 1 (EK1200)/Term 11 (EK1122)/Term 12 (EK1100)/Term 32 (EL7031)
//     Drive/Inputs/In/nState1 @bit 3 <-> STM Status/Status/Error
//     Drive/Inputs/In/nState1 @bit 5 <-> STM Status/Status/Moving negative
//     Drive/Inputs/In/nState1 @bit 4 <-> STM Status/Status/Moving positive
//     Drive/Inputs/In/nState1 @bit 1 <-> STM Status/Status/Ready
//     Drive/Inputs/In/nState1 <-> STM Status/Status/Ready to enable
//     Drive/Inputs/In/nState1 @bit 6 <-> STM Status/Status/Torque reduced
//     Drive/Inputs/In/nState1 @bit 2 <-> STM Status/Status/Warning
//     Drive/Inputs/In/nState2 @bit 3 <-> STM Status/Status/Digital input 1
//     Drive/Inputs/In/nState2 @bit 4 <-> STM Status/Status/Digital input 2
//     Drive/Inputs/In/nState2 @bit 5 <-> STM Status/Status/Sync error
//     Drive/Inputs/In/nState2 @bit 7 <-> STM Status/Status/TxPDO Toggle
//     Drive/Inputs/In/nState4 @bit 1 <-> WcState/InputToggle
//     Drive/Inputs/In/nState4 <-> WcState/WcState
//     Drive/Outputs/Out/nCtrl1 <-> STM Control/Control/Enable
//     Drive/Outputs/Out/nCtrl1 @bit 2 <-> STM Control/Control/Reduce torque
//     Drive/Outputs/Out/nCtrl1 @bit 1 <-> STM Control/Control/Reset
//     Drive/Outputs/Out/nDataOut2[0] <-> STM Velocity/Velocity
//     Enc/Inputs/In/nDataIn1[0] <-> ENC Status compact/Counter value
//     Enc/Inputs/In/nDataIn2[0] <-> ENC Status compact/Latch value
//     Enc/Inputs/In/nState1 @bit 4 <-> ENC Status compact/Status/Counter overflow
//     Enc/Inputs/In/nState1 @bit 3 <-> ENC Status compact/Status/Counter underflow
//     Enc/Inputs/In/nState1 @bit 1 <-> ENC Status compact/Status/Latch extern valid
//     Enc/Inputs/In/nState1 @bit 2 <-> ENC Status compact/Status/Set counter done
//     Enc/Inputs/In/nState2 @bit 4 <-> ENC Status compact/Status/Status of extern latch
//     Enc/Inputs/In/nState2 @bit 5 <-> ENC Status compact/Status/Sync error
//     Enc/Inputs/In/nState2 @bit 7 <-> ENC Status compact/Status/TxPDO Toggle
//     Enc/Inputs/In/nState4 @bit 1 <-> WcState/InputToggle
//     Enc/Inputs/In/nState4 <-> WcState/WcState
//     Enc/Outputs/Out/nCtrl1 @bit 3 <-> ENC Control compact/Control/Enable latch extern on negative edge
//     Enc/Outputs/Out/nCtrl1 @bit 1 <-> ENC Control compact/Control/Enable latch extern on positive edge
//     Enc/Outputs/Out/nCtrl1 @bit 2 <-> ENC Control compact/Control/Set counter
//     Enc/Outputs/Out/nDataOut1[0] <-> ENC Control compact/Set counter value
//   (this object) <-> Device 1 (EtherCAT)/Term 1 (EK1200)/Term 11 (EK1122)/Term 12 (EK1100)/Term 33 (EL7031)
//     Drive/Inputs/In/nState1 @bit 3 <-> STM Status/Status/Error
//     Drive/Inputs/In/nState1 @bit 5 <-> STM Status/Status/Moving negative
//     Drive/Inputs/In/nState1 @bit 4 <-> STM Status/Status/Moving positive
//     Drive/Inputs/In/nState1 @bit 1 <-> STM Status/Status/Ready
//     Drive/Inputs/In/nState1 <-> STM Status/Status/Ready to enable
//     Drive/Inputs/In/nState1 @bit 6 <-> STM Status/Status/Torque reduced
//     Drive/Inputs/In/nState1 @bit 2 <-> STM Status/Status/Warning
//     Drive/Inputs/In/nState2 @bit 3 <-> STM Status/Status/Digital input 1
//     Drive/Inputs/In/nState2 @bit 4 <-> STM Status/Status/Digital input 2
//     Drive/Inputs/In/nState2 @bit 5 <-> STM Status/Status/Sync error
//     Drive/Inputs/In/nState2 @bit 7 <-> STM Status/Status/TxPDO Toggle
//     Drive/Inputs/In/nState4 @bit 1 <-> WcState/InputToggle
//     Drive/Inputs/In/nState4 <-> WcState/WcState
//     Drive/Outputs/Out/nCtrl1 <-> STM Control/Control/Enable
//     Drive/Outputs/Out/nCtrl1 @bit 2 <-> STM Control/Control/Reduce torque
//     Drive/Outputs/Out/nCtrl1 @bit 1 <-> STM Control/Control/Reset
//     Drive/Outputs/Out/nDataOut2[0] <-> STM Velocity/Velocity
//     Enc/Inputs/In/nDataIn1[0] <-> ENC Status compact/Counter value
//     Enc/Inputs/In/nDataIn2[0] <-> ENC Status compact/Latch value
//     Enc/Inputs/In/nState1 @bit 4 <-> ENC Status compact/Status/Counter overflow
//     Enc/Inputs/In/nState1 @bit 3 <-> ENC Status compact/Status/Counter underflow
//     Enc/Inputs/In/nState1 @bit 1 <-> ENC Status compact/Status/Latch extern valid
//     Enc/Inputs/In/nState1 @bit 2 <-> ENC Status compact/Status/Set counter done
//     Enc/Inputs/In/nState2 @bit 4 <-> ENC Status compact/Status/Status of extern latch
//     Enc/Inputs/In/nState2 @bit 5 <-> ENC Status compact/Status/Sync error
//     Enc/Inputs/In/nState2 @bit 7 <-> ENC Status compact/Status/TxPDO Toggle
//     Enc/Inputs/In/nState4 @bit 1 <-> WcState/InputToggle
//     Enc/Inputs/In/nState4 <-> WcState/WcState
//     Enc/Outputs/Out/nCtrl1 @bit 3 <-> ENC Control compact/Control/Enable latch extern on negative edge
//     Enc/Outputs/Out/nCtrl1 @bit 1 <-> ENC Control compact/Control/Enable latch extern on positive edge
//     Enc/Outputs/Out/nCtrl1 @bit 2 <-> ENC Control compact/Control/Set counter
//     Enc/Outputs/Out/nDataOut1[0] <-> ENC Control compact/Set counter value
//   plc_polycap_01 Instance <-> Device 1 (EtherCAT)/Term 1 (EK1200)/POLYCAP1-EL1088-E4
//     PlcTask Inputs/Main.M{1..4}.bLimitBackwardEnable <-> Channel {2..8 step 2}/Input  (4 links)
//     PlcTask Inputs/Main.M{1..4}.bLimitForwardEnable <-> Channel {1..7 step 2}/Input  (4 links)
//   plc_polycap_01 Instance <-> Device 1 (EtherCAT)/Term 1 (EK1200)/POLYCAP1-EL1088-E9
//     PlcTask Inputs/Main.M5.bLimitBackwardEnable <-> Channel 2/Input
//     PlcTask Inputs/Main.M6.bLimitBackwardEnable <-> Channel 4/Input
//     PlcTask Inputs/Main.M5.bLimitForwardEnable <-> Channel 1/Input
//     PlcTask Inputs/Main.M6.bLimitForwardEnable <-> Channel 3/Input
//   plc_polycap_01 Instance <-> Device 1 (EtherCAT)/Term 1 (EK1200)/Term 11 (EK1122)/Term 12 (EK1100)/POLYCAP2-EL1088-E14
//     PlcTask Inputs/Main.M{15..18}.bLimitBackwardEnable <-> Channel {2..8 step 2}/Input  (4 links)
//     PlcTask Inputs/Main.M{15..18}.bLimitForwardEnable <-> Channel {1..7 step 2}/Input  (4 links)
//   plc_polycap_01 Instance <-> Device 1 (EtherCAT)/Term 1 (EK1200)/Term 11 (EK1122)/Term 12 (EK1100)/POLYCAP2-EL1088-E19
//     PlcTask Inputs/Main.M{19..22}.bLimitBackwardEnable <-> Channel {2..8 step 2}/Input  (4 links)
//     PlcTask Inputs/Main.M{19..22}.bLimitForwardEnable <-> Channel {1..7 step 2}/Input  (4 links)
//   plc_polycap_01 Instance <-> Device 1 (EtherCAT)/Term 1 (EK1200)/Term 11 (EK1122)/Term 12 (EK1100)/POLYCAP2-EL1088-E3
//     PlcTask Inputs/Main.M{7..10}.bLimitBackwardEnable <-> Channel {2..8 step 2}/Input  (4 links)
//     PlcTask Inputs/Main.M{7..10}.bLimitForwardEnable <-> Channel {1..7 step 2}/Input  (4 links)
//   plc_polycap_01 Instance <-> Device 1 (EtherCAT)/Term 1 (EK1200)/Term 11 (EK1122)/Term 12 (EK1100)/POLYCAP2-EL1088-E8
//     PlcTask Inputs/Main.M{11..14}.bLimitBackwardEnable <-> Channel {2..8 step 2}/Input  (4 links)
//     PlcTask Inputs/Main.M{11..14}.bLimitForwardEnable <-> Channel {1..7 step 2}/Input  (4 links)
//   plc_polycap_01 Instance <-> NC-Task 1 SAF/Axes/Axis 1 POLYCAP-DET-Z
//     PlcTask Inputs/Main.M1.Axis.NcToPlc <-> Outputs/ToPlc
//     PlcTask Outputs/Main.M1.Axis.PlcToNc <-> Inputs/FromPlc
//   plc_polycap_01 Instance <-> NC-Task 1 SAF/Axes/Axis 10 POLYCAP-CRY-S-X
//     PlcTask Inputs/Main.M10.Axis.NcToPlc <-> Outputs/ToPlc
//     PlcTask Outputs/Main.M10.Axis.PlcToNc <-> Inputs/FromPlc
//   plc_polycap_01 Instance <-> NC-Task 1 SAF/Axes/Axis 11 POLYCAP-CRY-M-SWI
//     PlcTask Inputs/Main.M11.Axis.NcToPlc <-> Outputs/ToPlc
//     PlcTask Outputs/Main.M11.Axis.PlcToNc <-> Inputs/FromPlc
//   plc_polycap_01 Instance <-> NC-Task 1 SAF/Axes/Axis 12 POLYCAP-CRY-M-X
//     PlcTask Inputs/Main.M12.Axis.NcToPlc <-> Outputs/ToPlc
//     PlcTask Outputs/Main.M12.Axis.PlcToNc <-> Inputs/FromPlc
//   plc_polycap_01 Instance <-> NC-Task 1 SAF/Axes/Axis 13 POLYCAP-CRY-S-ROT
//     PlcTask Inputs/Main.M13.Axis.NcToPlc <-> Outputs/ToPlc
//     PlcTask Outputs/Main.M13.Axis.PlcToNc <-> Inputs/FromPlc
//   plc_polycap_01 Instance <-> NC-Task 1 SAF/Axes/Axis 14 POLYCAP-CRY-S-Y
//     PlcTask Inputs/Main.M14.Axis.NcToPlc <-> Outputs/ToPlc
//     PlcTask Outputs/Main.M14.Axis.PlcToNc <-> Inputs/FromPlc
//   plc_polycap_01 Instance <-> NC-Task 1 SAF/Axes/Axis 15 POLYCAP-CRY-M-ROT
//     PlcTask Inputs/Main.M15.Axis.NcToPlc <-> Outputs/ToPlc
//     PlcTask Outputs/Main.M15.Axis.PlcToNc <-> Inputs/FromPlc
//   plc_polycap_01 Instance <-> NC-Task 1 SAF/Axes/Axis 16 POLYCAP-CRY-M-Y
//     PlcTask Inputs/Main.M16.Axis.NcToPlc <-> Outputs/ToPlc
//     PlcTask Outputs/Main.M16.Axis.PlcToNc <-> Inputs/FromPlc
//   plc_polycap_01 Instance <-> NC-Task 1 SAF/Axes/Axis 17 POLYCAP-PC-S-X
//     PlcTask Inputs/Main.M17.Axis.NcToPlc <-> Outputs/ToPlc
//     PlcTask Outputs/Main.M17.Axis.PlcToNc <-> Inputs/FromPlc
//   plc_polycap_01 Instance <-> NC-Task 1 SAF/Axes/Axis 18 POLYCAP-PC-S-Z
//     PlcTask Inputs/Main.M18.Axis.NcToPlc <-> Outputs/ToPlc
//     PlcTask Outputs/Main.M18.Axis.PlcToNc <-> Inputs/FromPlc
//   plc_polycap_01 Instance <-> NC-Task 1 SAF/Axes/Axis 19 POLYCAP-PC-M-X
//     PlcTask Inputs/Main.M19.Axis.NcToPlc <-> Outputs/ToPlc
//     PlcTask Outputs/Main.M19.Axis.PlcToNc <-> Inputs/FromPlc
//   plc_polycap_01 Instance <-> NC-Task 1 SAF/Axes/Axis 2 POLYCAP-CRY-N-SWI
//     PlcTask Inputs/Main.M2.Axis.NcToPlc <-> Outputs/ToPlc
//     PlcTask Outputs/Main.M2.Axis.PlcToNc <-> Inputs/FromPlc
//   plc_polycap_01 Instance <-> NC-Task 1 SAF/Axes/Axis 20 POLYCAP-PC-M-Z
//     PlcTask Inputs/Main.M20.Axis.NcToPlc <-> Outputs/ToPlc
//     PlcTask Outputs/Main.M20.Axis.PlcToNc <-> Inputs/FromPlc
//   plc_polycap_01 Instance <-> NC-Task 1 SAF/Axes/Axis 21 POLYCAP-PC-S-Y
//     PlcTask Inputs/Main.M21.Axis.NcToPlc <-> Outputs/ToPlc
//     PlcTask Outputs/Main.M21.Axis.PlcToNc <-> Inputs/FromPlc
//   plc_polycap_01 Instance <-> NC-Task 1 SAF/Axes/Axis 22 POLYCAP-PC-M-Y
//     PlcTask Inputs/Main.M22.Axis.NcToPlc <-> Outputs/ToPlc
//     PlcTask Outputs/Main.M22.Axis.PlcToNc <-> Inputs/FromPlc
//   plc_polycap_01 Instance <-> NC-Task 1 SAF/Axes/Axis 3 POLYCAP-CRY-N-X
//     PlcTask Inputs/Main.M3.Axis.NcToPlc <-> Outputs/ToPlc
//     PlcTask Outputs/Main.M3.Axis.PlcToNc <-> Inputs/FromPlc
//   plc_polycap_01 Instance <-> NC-Task 1 SAF/Axes/Axis 4 POLYCAP-CRY-N-ROT
//     PlcTask Inputs/Main.M4.Axis.NcToPlc <-> Outputs/ToPlc
//     PlcTask Outputs/Main.M4.Axis.PlcToNc <-> Inputs/FromPlc
//   plc_polycap_01 Instance <-> NC-Task 1 SAF/Axes/Axis 5 POLYCAP-CRY-N-Y
//     PlcTask Inputs/Main.M5.Axis.NcToPlc <-> Outputs/ToPlc
//     PlcTask Outputs/Main.M5.Axis.PlcToNc <-> Inputs/FromPlc
//   plc_polycap_01 Instance <-> NC-Task 1 SAF/Axes/Axis 6 POLYCAP-PC-N-X
//     PlcTask Inputs/Main.M6.Axis.NcToPlc <-> Outputs/ToPlc
//     PlcTask Outputs/Main.M6.Axis.PlcToNc <-> Inputs/FromPlc
//   plc_polycap_01 Instance <-> NC-Task 1 SAF/Axes/Axis 7 POLYCAP-PC-N-Z
//     PlcTask Inputs/Main.M7.Axis.NcToPlc <-> Outputs/ToPlc
//     PlcTask Outputs/Main.M7.Axis.PlcToNc <-> Inputs/FromPlc
//   plc_polycap_01 Instance <-> NC-Task 1 SAF/Axes/Axis 8 POLYCAP-PC-N-Y
//     PlcTask Inputs/Main.M8.Axis.NcToPlc <-> Outputs/ToPlc
//     PlcTask Outputs/Main.M8.Axis.PlcToNc <-> Inputs/FromPlc
//   plc_polycap_01 Instance <-> NC-Task 1 SAF/Axes/Axis 9 POLYCAP-CRY-S-SWI
//     PlcTask Inputs/Main.M9.Axis.NcToPlc <-> Outputs/ToPlc
//     PlcTask Outputs/Main.M9.Axis.PlcToNc <-> Inputs/FromPlc

// ---- GVLs/Main.TcGVL
{attribute 'qualified_only'}
VAR_GLOBAL

    // U/N North: 5 Axes
    {attribute 'pytmc' := 'pv: POLYCAP:DET:Z'}
    {attribute 'TcLinkTo' := '.bLimitForwardEnable  := TIIB[POLYCAP1-EL1088-E4]^Channel 1^Input;
                              .bLimitBackwardEnable := TIIB[POLYCAP1-EL1088-E4]^Channel 2^Input'}
    M1: DUT_MotionStage := (sName := 'POLYCAP:DET:Z');

    {attribute 'pytmc' := 'pv: POLYCAP:CRY:N:SWI'}
    {attribute 'TcLinkTo' := '.bLimitForwardEnable  := TIIB[POLYCAP1-EL1088-E4]^Channel 3^Input;
                              .bLimitBackwardEnable := TIIB[POLYCAP1-EL1088-E4]^Channel 4^Input'}
    M2: DUT_MotionStage := (sName := 'POLYCAP:CRY:N:SWI');

    {attribute 'pytmc' := 'pv: POLYCAP:CRY:N:X'}
    {attribute 'TcLinkTo' := '.bLimitForwardEnable  := TIIB[POLYCAP1-EL1088-E4]^Channel 5^Input;
                              .bLimitBackwardEnable := TIIB[POLYCAP1-EL1088-E4]^Channel 6^Input'}
    M3: DUT_MotionStage := (sName := 'POLYCAP:CRY:N:X');

    {attribute 'pytmc' := 'pv: POLYCAP:CRY:N:ROT'}
    {attribute 'TcLinkTo' := '.bLimitForwardEnable  := TIIB[POLYCAP1-EL1088-E4]^Channel 7^Input;
                              .bLimitBackwardEnable := TIIB[POLYCAP1-EL1088-E4]^Channel 8^Input'}
    M4: DUT_MotionStage := (sName := 'POLYCAP:CRY:N:ROT');

    {attribute 'pytmc' := 'pv: POLYCAP:CRY:N:Y'}
    {attribute 'TcLinkTo' := '.bLimitForwardEnable  := TIIB[POLYCAP1-EL1088-E9]^Channel 1^Input;
                              .bLimitBackwardEnable := TIIB[POLYCAP1-EL1088-E9]^Channel 2^Input'}
    M5: DUT_MotionStage := (sName := 'POLYCAP:CRY:N:Y');

    // D/N North: 3 Axes
    {attribute 'pytmc' := 'pv: POLYCAP:PC:N:X'}
    {attribute 'TcLinkTo' := '.bLimitForwardEnable  := TIIB[POLYCAP1-EL1088-E9]^Channel 3^Input;
                              .bLimitBackwardEnable := TIIB[POLYCAP1-EL1088-E9]^Channel 4^Input'}
    M6: DUT_MotionStage := (sName := 'POLYCAP:PC:N:X');

    {attribute 'pytmc' := 'pv: POLYCAP:PC:N:Z'}
    {attribute 'TcLinkTo' := '.bLimitForwardEnable  := TIIB[POLYCAP2-EL1088-E3]^Channel 1^Input;
                              .bLimitBackwardEnable := TIIB[POLYCAP2-EL1088-E3]^Channel 2^Input'}
    M7: DUT_MotionStage := (sName := 'POLYCAP:PC:N:Z');

    {attribute 'pytmc' := 'pv: POLYCAP:PC:N:Y'}
    {attribute 'TcLinkTo' := '.bLimitForwardEnable  := TIIB[POLYCAP2-EL1088-E3]^Channel 3^Input;
                              .bLimitBackwardEnable := TIIB[POLYCAP2-EL1088-E3]^Channel 4^Input'}
    M8: DUT_MotionStage := (sName := 'POLYCAP:PC:N:Y');

    // U/s South: 8 Axes

    {attribute 'pytmc' := 'pv: POLYCAP:CRY:S:SWI'}
    {attribute 'TcLinkTo' := '.bLimitForwardEnable  := TIIB[POLYCAP2-EL1088-E3]^Channel 5^Input;
                              .bLimitBackwardEnable := TIIB[POLYCAP2-EL1088-E3]^Channel 6^Input'}
    M9: DUT_MotionStage := (sName := 'POLYCAP:CRY:S:SWI');

    {attribute 'pytmc' := 'pv: POLYCAP:CRY:S:X'}
    {attribute 'TcLinkTo' := '.bLimitForwardEnable  := TIIB[POLYCAP2-EL1088-E3]^Channel 7^Input;
                              .bLimitBackwardEnable := TIIB[POLYCAP2-EL1088-E3]^Channel 8^Input'}
    M10: DUT_MotionStage := (sName := 'POLYCAP:CRY:S:X');

    {attribute 'pytmc' := 'pv: POLYCAP:CRY:M:SWI'}
    {attribute 'TcLinkTo' := '.bLimitForwardEnable  := TIIB[POLYCAP2-EL1088-E8]^Channel 1^Input;
                              .bLimitBackwardEnable := TIIB[POLYCAP2-EL1088-E8]^Channel 2^Input'}
    M11: DUT_MotionStage := (sName := 'POLYCAP:CRY:M:SWI');

    {attribute 'pytmc' := 'pv: POLYCAP:CRY:M:X'}
    {attribute 'TcLinkTo' := '.bLimitForwardEnable  := TIIB[POLYCAP2-EL1088-E8]^Channel 3^Input;
                              .bLimitBackwardEnable := TIIB[POLYCAP2-EL1088-E8]^Channel 4^Input'}
    M12: DUT_MotionStage := (sName := 'POLYCAP:CRY:M:X');

    {attribute 'pytmc' := 'pv: POLYCAP:CRY:S:ROT'}
    {attribute 'TcLinkTo' := '.bLimitForwardEnable  := TIIB[POLYCAP2-EL1088-E8]^Channel 5^Input;
                              .bLimitBackwardEnable := TIIB[POLYCAP2-EL1088-E8]^Channel 6^Input'}
    M13: DUT_MotionStage := (sName := 'POLYCAP:CRY:S:ROT');

    {attribute 'pytmc' := 'pv: POLYCAP:CRY:S:Y'}
    {attribute 'TcLinkTo' := '.bLimitForwardEnable  := TIIB[POLYCAP2-EL1088-E8]^Channel 7^Input;
                              .bLimitBackwardEnable := TIIB[POLYCAP2-EL1088-E8]^Channel 8^Input'}
    M14: DUT_MotionStage := (sName := 'POLYCAP:CRY:S:Y');

    {attribute 'pytmc' := 'pv: POLYCAP:CRY:M:ROT'}
    {attribute 'TcLinkTo' := '.bLimitForwardEnable  := TIIB[POLYCAP2-EL1088-E14]^Channel 1^Input;
                              .bLimitBackwardEnable := TIIB[POLYCAP2-EL1088-E14]^Channel 2^Input'}
    M15: DUT_MotionStage := (sName := 'POLYCAP:CRY:M:ROT');

    {attribute 'pytmc' := 'pv: POLYCAP:CRY:M:Y'}
    {attribute 'TcLinkTo' := '.bLimitForwardEnable  := TIIB[POLYCAP2-EL1088-E14]^Channel 3^Input;
                              .bLimitBackwardEnable := TIIB[POLYCAP2-EL1088-E14]^Channel 4^Input'}
    M16: DUT_MotionStage := (sName := 'POLYCAP:CRY:M:Y');

    // D/S South: 6 Axes


    {attribute 'pytmc' := 'pv: POLYCAP:PC:S:X'}
    {attribute 'TcLinkTo' := '.bLimitForwardEnable  := TIIB[POLYCAP2-EL1088-E14]^Channel 5^Input;
                              .bLimitBackwardEnable := TIIB[POLYCAP2-EL1088-E14]^Channel 6^Input'}
    M17: DUT_MotionStage := (sName := 'POLYCAP:PC:S:X');


    {attribute 'pytmc' := 'pv: POLYCAP:PC:S:Z'}
    {attribute 'TcLinkTo' := '.bLimitForwardEnable  := TIIB[POLYCAP2-EL1088-E14]^Channel 7^Input;
                              .bLimitBackwardEnable := TIIB[POLYCAP2-EL1088-E14]^Channel 8^Input'}
    M18: DUT_MotionStage := (sName := 'POLYCAP:PC:S:Z');


    {attribute 'pytmc' := 'pv: POLYCAP:PC:M:X'}
    {attribute 'TcLinkTo' := '.bLimitForwardEnable  := TIIB[POLYCAP2-EL1088-E19]^Channel 1^Input;
                              .bLimitBackwardEnable := TIIB[POLYCAP2-EL1088-E19]^Channel 2^Input'}
    M19: DUT_MotionStage := (sName := 'POLYCAP:PC:M:X');


    {attribute 'pytmc' := 'pv: POLYCAP:PC:M:Z'}
    {attribute 'TcLinkTo' := '.bLimitForwardEnable  := TIIB[POLYCAP2-EL1088-E19]^Channel 3^Input;
                              .bLimitBackwardEnable := TIIB[POLYCAP2-EL1088-E19]^Channel 4^Input'}
    M20: DUT_MotionStage := (sName := 'POLYCAP:PC:M:Z');


    {attribute 'pytmc' := 'pv: POLYCAP:PC:S:Y'}
    {attribute 'TcLinkTo' := '.bLimitForwardEnable  := TIIB[POLYCAP2-EL1088-E19]^Channel 5^Input;
                              .bLimitBackwardEnable := TIIB[POLYCAP2-EL1088-E19]^Channel 6^Input'}
    M21: DUT_MotionStage := (sName := 'POLYCAP:PC:S:Y');


    {attribute 'pytmc' := 'pv: POLYCAP:PC:M:Y'}
    {attribute 'TcLinkTo' := '.bLimitForwardEnable  := TIIB[POLYCAP2-EL1088-E19]^Channel 7^Input;
                              .bLimitBackwardEnable := TIIB[POLYCAP2-EL1088-E19]^Channel 8^Input'}
    M22: DUT_MotionStage := (sName := 'POLYCAP:PC:M:Y');



END_VAR

// ---- POUs/PRG_SPEC.TcPOU
PROGRAM PRG_SPEC
VAR
    fbPOLYCAP_DET_Z: FB_MotionStage;
    fbPOLYCAP_CRY_N_SWI: FB_MotionStage;
    fbPOLYCAP_CRY_N_X: FB_MotionStage;
    fbPOLYCAP_CRY_N_ROT: FB_MotionStage;
    fbPOLYCAP_CRY_N_Y: FB_MotionStage;
    fbPOLYCAP_PC_N_X: FB_MotionStage;
    fbPOLYCAP_PC_N_Z: FB_MotionStage;
    fbPOLYCAP_PC_N_Y: FB_MotionStage;
    fbPOLYCAP_CRY_S_SWI: FB_MotionStage;
    fbPOLYCAP_CRY_S_X: FB_MotionStage;
    fbPOLYCAP_CRY_M_SWI: FB_MotionStage;
    fbPOLYCAP_CRY_M_X: FB_MotionStage;
    fbPOLYCAP_CRY_S_ROT: FB_MotionStage;
    fbPOLYCAP_CRY_S_Y: FB_MotionStage;
    fbPOLYCAP_CRY_M_ROT: FB_MotionStage;
    fbPOLYCAP_CRY_M_Y: FB_MotionStage;
    fbPOLYCAP_PC_S_X: FB_MotionStage;
    fbPOLYCAP_PC_S_Z: FB_MotionStage;
    fbPOLYCAP_PC_M_X: FB_MotionStage;
    fbPOLYCAP_PC_M_Z: FB_MotionStage;
    fbPOLYCAP_PC_S_Y: FB_MotionStage;
    fbPOLYCAP_PC_M_Y: FB_MotionStage;
    stMotionStage: INT;


    // Only do some of the puts on init
    bInit: BOOL := FALSE;

END_VAR

fbPOLYCAP_DET_Z(stMotionStage:=Main.M1);
fbPOLYCAP_CRY_N_SWI(stMotionStage:=Main.M2);
fbPOLYCAP_CRY_N_X(stMotionStage:=Main.M3);
fbPOLYCAP_CRY_N_ROT(stMotionStage:=Main.M4);
fbPOLYCAP_CRY_N_Y(stMotionStage:=Main.M5);
fbPOLYCAP_PC_N_X(stMotionStage:=Main.M6);
fbPOLYCAP_PC_N_Z(stMotionStage:=Main.M7);
fbPOLYCAP_PC_N_Y(stMotionStage:=Main.M8);
fbPOLYCAP_CRY_S_SWI(stMotionStage:=Main.M9);
fbPOLYCAP_CRY_S_X(stMotionStage:=Main.M10);
fbPOLYCAP_CRY_M_SWI(stMotionStage:=Main.M11);
fbPOLYCAP_CRY_M_X(stMotionStage:=Main.M12);
fbPOLYCAP_CRY_S_ROT(stMotionStage:=Main.M13);
fbPOLYCAP_CRY_S_Y(stMotionStage:=Main.M14);
fbPOLYCAP_CRY_M_ROT(stMotionStage:=Main.M15);
fbPOLYCAP_CRY_M_Y(stMotionStage:=Main.M16);
fbPOLYCAP_PC_S_X(stMotionStage:=Main.M17);
fbPOLYCAP_PC_S_Z(stMotionStage:=Main.M18);
fbPOLYCAP_PC_M_X(stMotionStage:=Main.M19);
fbPOLYCAP_PC_M_Z(stMotionStage:=Main.M20);
fbPOLYCAP_PC_S_Y(stMotionStage:=Main.M21);
fbPOLYCAP_PC_M_Y(stMotionStage:=Main.M22);








IF NOT bInit THEN // Easier to debug if you can write to these
    Main.M1.bHardwareEnable := TRUE;
    Main.M1.bPowerSelf := TRUE;
    Main.M1.nEnableMode := ENUM_StageEnableMode.DURING_MOTION;
//	Main.M1.nHomingMode := ENUM_EpicsHomeCmd.LOW_LIMIT;
//	Main.M1.nEnableMode := ENUM_StageEnableMode.ALWAYS;

    Main.M2.bHardwareEnable := TRUE;
    Main.M2.bPowerSelf := TRUE;
    Main.M2.nEnableMode := ENUM_StageEnableMode.DURING_MOTION;
//	Main.M2.nHomingMode := ENUM_EpicsHomeCmd.LOW_LIMIT;
//	Main.M2.nEnableMode := ENUM_StageEnableMode.ALWAYS;

    Main.M3.bHardwareEnable := TRUE;
    Main.M3.bPowerSelf := TRUE;
    Main.M3.nEnableMode := ENUM_StageEnableMode.DURING_MOTION;
//	Main.M3.nHomingMode := ENUM_EpicsHomeCmd.LOW_LIMIT;
//	Main.M3.nEnableMode := ENUM_StageEnableMode.ALWAYS;

    Main.M4.bHardwareEnable := TRUE;
    Main.M4.bPowerSelf := TRUE;
    Main.M4.nEnableMode := ENUM_StageEnableMode.DURING_MOTION;
//	Main.M4.nHomingMode := ENUM_EpicsHomeCmd.LOW_LIMIT;
//	Main.M4.nEnableMode := ENUM_StageEnableMode.ALWAYS;


    Main.M5.bHardwareEnable := TRUE;
    Main.M5.bPowerSelf := TRUE;
    Main.M5.nEnableMode := ENUM_StageEnableMode.DURING_MOTION;
//	Main.M5.nHomingMode := ENUM_EpicsHomeCmd.LOW_LIMIT;
//	Main.M5.nEnableMode := ENUM_StageEnableMode.ALWAYS;

    Main.M6.bHardwareEnable := TRUE;
    Main.M6.bPowerSelf := TRUE;
    Main.M6.nEnableMode := ENUM_StageEnableMode.DURING_MOTION;
//	Main.M6.nHomingMode := ENUM_EpicsHomeCmd.LOW_LIMIT;
//	Main.M6.nEnableMode := ENUM_StageEnableMode.ALWAYS;

    Main.M7.bHardwareEnable := TRUE;
    Main.M7.bPowerSelf := TRUE;
    Main.M7.nEnableMode := ENUM_StageEnableMode.DURING_MOTION;
//	Main.M7.nHomingMode := ENUM_EpicsHomeCmd.LOW_LIMIT;
//	Main.M7.nEnableMode := ENUM_StageEnableMode.ALWAYS;

    Main.M8.bHardwareEnable := TRUE;
    Main.M8.bPowerSelf := TRUE;
    Main.M8.nEnableMode := ENUM_StageEnableMode.DURING_MOTION;
//	Main.M8.nHomingMode := ENUM_EpicsHomeCmd.LOW_LIMIT;
//	Main.M8.nEnableMode := ENUM_StageEnableMode.ALWAYS;

    Main.M9.bHardwareEnable := TRUE;
    Main.M9.bPowerSelf := TRUE;
    Main.M9.nEnableMode := ENUM_StageEnableMode.DURING_MOTION;
//	Main.M9.nHomingMode := ENUM_EpicsHomeCmd.LOW_LIMIT;
//	Main.M9.nEnableMode := ENUM_StageEnableMode.ALWAYS;

    Main.M10.bHardwareEnable := TRUE;
    Main.M10.bPowerSelf := TRUE;
    Main.M10.nEnableMode := ENUM_StageEnableMode.DURING_MOTION;
//	Main.M10.nHomingMode := ENUM_EpicsHomeCmd.LOW_LIMIT;
//	Main.M10.nEnableMode := ENUM_StageEnableMode.ALWAYS;

    Main.M11.bHardwareEnable := TRUE;
    Main.M11.bPowerSelf := TRUE;
    Main.M11.nEnableMode := ENUM_StageEnableMode.DURING_MOTION;
//	Main.M11.nHomingMode := ENUM_EpicsHomeCmd.LOW_LIMIT;
//	Main.M11.nEnableMode := ENUM_StageEnableMode.ALWAYS;

    Main.M12.bHardwareEnable := TRUE;
    Main.M12.bPowerSelf := TRUE;
    Main.M12.nEnableMode := ENUM_StageEnableMode.DURING_MOTION;
//	Main.M12.nHomingMode := ENUM_EpicsHomeCmd.LOW_LIMIT;
//	Main.M12.nEnableMode := ENUM_StageEnableMode.ALWAYS;

    Main.M13.bHardwareEnable := TRUE;
    Main.M13.bPowerSelf := TRUE;
    Main.M13.nEnableMode := ENUM_StageEnableMode.DURING_MOTION;
//	Main.M13.nHomingMode := ENUM_EpicsHomeCmd.LOW_LIMIT;
//	Main.M13.nEnableMode := ENUM_StageEnableMode.ALWAYS;

    Main.M14.bHardwareEnable := TRUE;
    Main.M14.bPowerSelf := TRUE;
    Main.M14.nEnableMode := ENUM_StageEnableMode.DURING_MOTION;
//	Main.M14.nHomingMode := ENUM_EpicsHomeCmd.LOW_LIMIT;
//	Main.M14.nEnableMode := ENUM_StageEnableMode.ALWAYS;

    Main.M15.bHardwareEnable := TRUE;
    Main.M15.bPowerSelf := TRUE;
    Main.M15.nEnableMode := ENUM_StageEnableMode.DURING_MOTION;
//	Main.M15.nHomingMode := ENUM_EpicsHomeCmd.LOW_LIMIT;
//	Main.M15.nEnableMode := ENUM_StageEnableMode.ALWAYS;

    Main.M16.bHardwareEnable := TRUE;
    Main.M16.bPowerSelf := TRUE;
    Main.M16.nEnableMode := ENUM_StageEnableMode.DURING_MOTION;
//	Main.M16.nHomingMode := ENUM_EpicsHomeCmd.LOW_LIMIT;
//	Main.M16.nEnableMode := ENUM_StageEnableMode.ALWAYS;

    Main.M17.bHardwareEnable := TRUE;
    Main.M17.bPowerSelf := TRUE;
    Main.M17.nEnableMode := ENUM_StageEnableMode.DURING_MOTION;
//	Main.M17.nHomingMode := ENUM_EpicsHomeCmd.LOW_LIMIT;
//	Main.M17.nEnableMode := ENUM_StageEnableMode.ALWAYS;

    Main.M18.bHardwareEnable := TRUE;
    Main.M18.bPowerSelf := TRUE;
    Main.M18.nEnableMode := ENUM_StageEnableMode.DURING_MOTION;
//	Main.M18.nHomingMode := ENUM_EpicsHomeCmd.LOW_LIMIT;
//	Main.M18.nEnableMode := ENUM_StageEnableMode.ALWAYS;

    Main.M19.bHardwareEnable := TRUE;
    Main.M19.bPowerSelf := TRUE;
    Main.M19.nEnableMode := ENUM_StageEnableMode.DURING_MOTION;
//	Main.M19.nHomingMode := ENUM_EpicsHomeCmd.LOW_LIMIT;
//	Main.M19.nEnableMode := ENUM_StageEnableMode.ALWAYS;

    Main.M20.bHardwareEnable := TRUE;
    Main.M20.bPowerSelf := TRUE;
    Main.M20.nEnableMode := ENUM_StageEnableMode.DURING_MOTION;
//	Main.M20.nHomingMode := ENUM_EpicsHomeCmd.LOW_LIMIT;
//	Main.M20.nEnableMode := ENUM_StageEnableMode.ALWAYS;

    Main.M21.bHardwareEnable := TRUE;
    Main.M21.bPowerSelf := TRUE;
    Main.M21.nEnableMode := ENUM_StageEnableMode.DURING_MOTION;
//	Main.M21.nHomingMode := ENUM_EpicsHomeCmd.LOW_LIMIT;
//	Main.M21.nEnableMode := ENUM_StageEnableMode.ALWAYS;

    Main.M22.bHardwareEnable := TRUE;
    Main.M22.bPowerSelf := TRUE;
    Main.M22.nEnableMode := ENUM_StageEnableMode.DURING_MOTION;
//	Main.M22.nHomingMode := ENUM_EpicsHomeCmd.LOW_LIMIT;
//	Main.M22.nEnableMode := ENUM_StageEnableMode.ALWAYS;

    bInit := True;
END_IF

END_PROGRAM
